ABB RAPID module: P104.mod

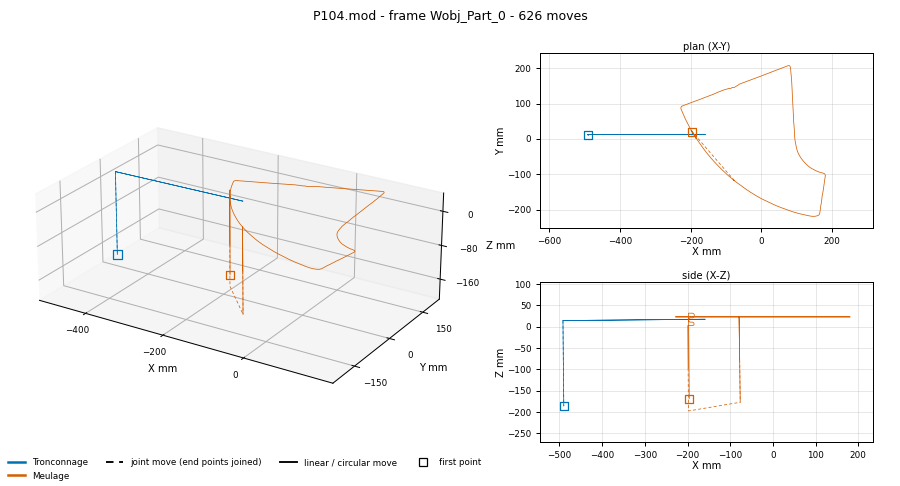
[picture p0: tool path of P104.mod in frame Wobj_Part_0, 626 of 631 moves have a stored position in this frame; points joined in program order, loops and branches not executed]
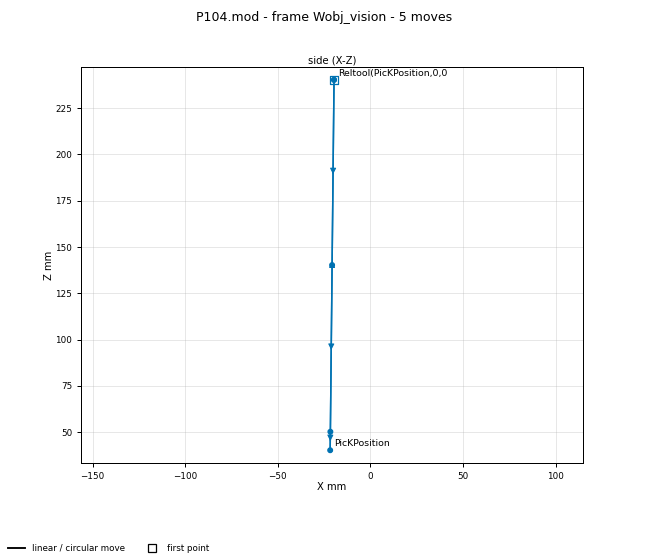
[picture p1: tool path of P104.mod in frame Wobj_vision, 5 of 631 moves have a stored position in this frame; points joined in program order, loops and branches not executed]
MODULE P104

    ! Nom         :P104
    ! Description :
    ! Créé le     :03/04/2023 16:24:55

    LOCAL CONST SPEEDDATA VitesseLente :=[10,500,0,0];
	LOCAL CONST SPEEDDATA VitesseRapide :=[30,500,0,0];
    !
    !Point de prise
    LOCAL PERS Robtarget PicKPosition := [[-21.7405517614,13.3135132251341,40.2938438381467],[-0.00337713641881813,-0.940755559571221,0.33904158472546,0.00428671346086143],[0,0,0,0],[8.999999E+09,8.999999E+09,8.999999E+09,8.999999E+09,8.999999E+09,8.999999E+09]];
	LOCAL PERS Pose Ref := [[0,0,0],[1,0,0,0]];
    !
    !Declaration des points de meulage

    !Tr_meulage_motif_1 : Meulage d'un motif
    LOCAL CONST Robtarget Tr_meulage_motif_1_0 := [[-197.52953125,22.28647265625,31.672755859375],[0.999972798976242,-0.00614910498762201,-0.0040037244179501,-0.000748335657728133],[0,0,0,0],[8.999999E+09,8.999999E+09,8.999999E+09,8.999999E+09,8.999999E+09,8.999999E+09]];
    LOCAL CONST Robtarget Tr_meulage_motif_1_1 := [[-196.9945,21.441646484375,31.672755859375],[0.999972798976242,-0.00614910498762201,-0.0040037244179501,-0.000748335657728133],[0,0,0,0],[8.999999E+09,8.999999E+09,8.999999E+09,8.999999E+09,8.999999E+09,8.999999E+09]];
    LOCAL CONST Robtarget Tr_meulage_motif_1_2 := [[-196.459453125,20.5968203125,31.6727578125],[0.999972798976242,-0.00614910498762201,-0.0040037244179501,-0.000748335657728133],[0,0,0,0],[8.999999E+09,8.999999E+09,8.999999E+09,8.999999E+09,8.999999E+09,8.999999E+09]];
    LOCAL CONST Robtarget Tr_meulage_motif_1_3 := [[-195.92440625,19.75199609375,31.6727578125],[0.999972798976242,-0.00614910498762201,-0.0040037244179501,-0.000748335657728133],[0,0,0,0],[8.999999E+09,8.999999E+09,8.999999E+09,8.999999E+09,8.999999E+09,8.999999E+09]];
    LOCAL CONST Robtarget Tr_meulage_motif_1_4 := [[-195.389375,18.907169921875,31.6727578125],[0.999972798976242,-0.00614910498762201,-0.0040037244179501,-0.000748335657728133],[0,0,0,0],[8.999999E+09,8.999999E+09,8.999999E+09,8.999999E+09,8.999999E+09,8.999999E+09]];
    LOCAL CONST Robtarget Tr_meulage_motif_1_5 := [[-194.854328125,18.06234375,31.672759765625],[0.999972798976242,-0.00614910498762201,-0.0040037244179501,-0.000748335657728133],[0,0,0,0],[8.999999E+09,8.999999E+09,8.999999E+09,8.999999E+09,8.999999E+09,8.999999E+09]];
    LOCAL CONST Robtarget Tr_meulage_motif_1_6 := [[-194.31928125,17.217517578125,31.672759765625],[0.999972798976242,-0.00614910498762201,-0.0040037244179501,-0.000748335657728133],[0,0,0,0],[8.999999E+09,8.999999E+09,8.999999E+09,8.999999E+09,8.999999E+09,8.999999E+09]];
    LOCAL CONST Robtarget Tr_meulage_motif_1_7 := [[-193.78425,16.3726923828125,31.672759765625],[0.999972798976242,-0.00614910498762201,-0.0040037244179501,-0.000748335657728133],[0,0,0,0],[8.999999E+09,8.999999E+09,8.999999E+09,8.999999E+09,8.999999E+09,8.999999E+09]];
    LOCAL CONST Robtarget Tr_meulage_motif_1_8 := [[-193.249203125,15.5278671875,31.67276171875],[0.999972798976242,-0.00614910498762201,-0.0040037244179501,-0.000748335657728133],[0,0,0,0],[8.999999E+09,8.999999E+09,8.999999E+09,8.999999E+09,8.999999E+09,8.999999E+09]];
    LOCAL CONST Robtarget Tr_meulage_motif_1_9 := [[-192.71415625,14.683041015625,31.67276171875],[0.999972798976242,-0.00614910498762201,-0.0040037244179501,-0.000748335657728133],[0,0,0,0],[8.999999E+09,8.999999E+09,8.999999E+09,8.999999E+09,8.999999E+09,8.999999E+09]];
    LOCAL CONST Robtarget Tr_meulage_motif_1_10 := [[-192.179125,13.8382158203125,31.67276171875],[0.999972798976242,-0.00614910498762201,-0.0040037244179501,-0.000748335657728133],[0,0,0,0],[8.999999E+09,8.999999E+09,8.999999E+09,8.999999E+09,8.999999E+09,8.999999E+09]];
    LOCAL CONST Robtarget Tr_meulage_motif_1_11 := [[-191.644078125,12.9933896484375,31.672763671875],[0.999972798976242,-0.00614910498762201,-0.0040037244179501,-0.000748335657728133],[0,0,0,0],[8.999999E+09,8.999999E+09,8.999999E+09,8.999999E+09,8.999999E+09,8.999999E+09]];
    LOCAL CONST Robtarget Tr_meulage_motif_1_12 := [[-191.10903125,12.148564453125,31.672763671875],[0.999972798976242,-0.00614910498762201,-0.0040037244179501,-0.000748335657728133],[0,0,0,0],[8.999999E+09,8.999999E+09,8.999999E+09,8.999999E+09,8.999999E+09,8.999999E+09]];
    LOCAL CONST Robtarget Tr_meulage_motif_1_13 := [[-190.574,11.30373828125,31.672763671875],[0.999972798976242,-0.00614910498762201,-0.0040037244179501,-0.000748335657728133],[0,0,0,0],[8.999999E+09,8.999999E+09,8.999999E+09,8.999999E+09,8.999999E+09,8.999999E+09]];
    LOCAL CONST Robtarget Tr_meulage_motif_1_14 := [[-190.038953125,10.4589130859375,31.672765625],[0.999972798976242,-0.00614910498762201,-0.0040037244179501,-0.000748335657728133],[0,0,0,0],[8.999999E+09,8.999999E+09,8.999999E+09,8.999999E+09,8.999999E+09,8.999999E+09]];
    LOCAL CONST Robtarget Tr_meulage_motif_1_15 := [[-189.50390625,9.6140869140625,31.672765625],[0.999972798976242,-0.00614910498762201,-0.0040037244179501,-0.000748335657728133],[0,0,0,0],[8.999999E+09,8.999999E+09,8.999999E+09,8.999999E+09,8.999999E+09,8.999999E+09]];
    LOCAL CONST Robtarget Tr_meulage_motif_1_16 := [[-188.968875,8.76926171875,31.672765625],[0.999972798976242,-0.00614910498762201,-0.0040037244179501,-0.000748335657728133],[0,0,0,0],[8.999999E+09,8.999999E+09,8.999999E+09,8.999999E+09,8.999999E+09,8.999999E+09]];
    LOCAL CONST Robtarget Tr_meulage_motif_1_17 := [[-188.433828125,7.92443603515625,31.672767578125],[0.999972798976242,-0.00614910498762201,-0.0040037244179501,-0.000748335657728133],[0,0,0,0],[8.999999E+09,8.999999E+09,8.999999E+09,8.999999E+09,8.999999E+09,8.999999E+09]];
    LOCAL CONST Robtarget Tr_meulage_motif_1_18 := [[-187.89878125,7.0796103515625,31.672767578125],[0.999972798976242,-0.00614910498762201,-0.0040037244179501,-0.000748335657728133],[0,0,0,0],[8.999999E+09,8.999999E+09,8.999999E+09,8.999999E+09,8.999999E+09,8.999999E+09]];
    LOCAL CONST Robtarget Tr_meulage_motif_1_19 := [[-187.368796875,6.24039208984375,31.562181640625],[0.999972798976242,-0.00614910498762201,-0.0040037244179501,-0.000748335657728133],[0,0,0,0],[8.999999E+09,8.999999E+09,8.999999E+09,8.999999E+09,8.999999E+09,8.999999E+09]];
    LOCAL CONST Robtarget Tr_meulage_motif_1_20 := [[-186.86440625,5.4394736328125,31.351009765625],[0.999972798976242,-0.00614910498762201,-0.0040037244179501,-0.000748335657728133],[0,0,0,0],[8.999999E+09,8.999999E+09,8.999999E+09,8.999999E+09,8.999999E+09,8.999999E+09]];
    LOCAL CONST Robtarget Tr_meulage_motif_1_21 := [[-186.410796875,4.71741357421875,31.07918359375],[0.999972798976242,-0.00614910498762201,-0.0040037244179501,-0.000748335657728133],[0,0,0,0],[8.999999E+09,8.999999E+09,8.999999E+09,8.999999E+09,8.999999E+09,8.999999E+09]];
    LOCAL CONST Robtarget Tr_meulage_motif_1_22 := [[-186.012203125,4.08216088867187,30.803263671875],[0.999972798976242,-0.00614910498762201,-0.0040037244179501,-0.000748335657728133],[0,0,0,0],[8.999999E+09,8.999999E+09,8.999999E+09,8.999999E+09,8.999999E+09,8.999999E+09]];
    LOCAL CONST Robtarget Tr_meulage_motif_1_23 := [[-185.42903125,3.148189453125,30.1871796875],[0.999972798976242,-0.00614910498762201,-0.0040037244179501,-0.000748335657728133],[0,0,0,0],[8.999999E+09,8.999999E+09,8.999999E+09,8.999999E+09,8.999999E+09,8.999999E+09]];
    LOCAL CONST Robtarget Tr_meulage_motif_1_24 := [[-184.88940625,2.27801293945312,29.339580078125],[0.999972798976242,-0.00614910498762201,-0.0040037244179501,-0.000748335657728133],[0,0,0,0],[8.999999E+09,8.999999E+09,8.999999E+09,8.999999E+09,8.999999E+09,8.999999E+09]];
    LOCAL CONST Robtarget Tr_meulage_motif_1_25 := [[-184.44575,1.55563366699219,28.315771484375],[0.999972798976242,-0.00614910498762201,-0.0040037244179501,-0.000748335657728133],[0,0,0,0],[8.999999E+09,8.999999E+09,8.999999E+09,8.999999E+09,8.999999E+09,8.999999E+09]];
    LOCAL CONST Robtarget Tr_meulage_motif_1_26 := [[-184.195328125,1.13640502929688,27.199658203125],[0.999972798976242,-0.00614910498762201,-0.0040037244179501,-0.000748335657728133],[0,0,0,0],[8.999999E+09,8.999999E+09,8.999999E+09,8.999999E+09,8.999999E+09,8.999999E+09]];
    LOCAL CONST Robtarget Tr_meulage_motif_1_27 := [[-184.187578125,1.10928845214844,26.503734375],[0.999972798976242,-0.00614910498762201,-0.0040037244179501,-0.000748335657728133],[0,0,0,0],[8.999999E+09,8.999999E+09,8.999999E+09,8.999999E+09,8.999999E+09,8.999999E+09]];
    LOCAL CONST Robtarget Tr_meulage_motif_1_28 := [[-184.193953125,1.10524719238281,25.84252734375],[0.999972798976242,-0.00614910498762201,-0.0040037244179501,-0.000748335657728133],[0,0,0,0],[8.999999E+09,8.999999E+09,8.999999E+09,8.999999E+09,8.999999E+09,8.999999E+09]];
    LOCAL CONST Robtarget Tr_meulage_motif_1_29 := [[-184.2296875,1.14756665039062,25.1814765625],[0.999972798976242,-0.00614910498762201,-0.0040037244179501,-0.000748335657728133],[0,0,0,0],[8.999999E+09,8.999999E+09,8.999999E+09,8.999999E+09,8.999999E+09,8.999999E+09]];
    LOCAL CONST Robtarget Tr_meulage_motif_1_30 := [[-184.506890625,1.5617412109375,24.079798828125],[0.999972798976242,-0.00614910498762201,-0.0040037244179501,-0.000748335657728133],[0,0,0,0],[8.999999E+09,8.999999E+09,8.999999E+09,8.999999E+09,8.999999E+09,8.999999E+09]];
    LOCAL CONST Robtarget Tr_meulage_motif_1_31 := [[-184.9749375,2.27928784179687,23.07323828125],[0.999972798976242,-0.00614910498762201,-0.0040037244179501,-0.000748335657728133],[0,0,0,0],[8.999999E+09,8.999999E+09,8.999999E+09,8.999999E+09,8.999999E+09,8.999999E+09]];
    LOCAL CONST Robtarget Tr_meulage_motif_1_32 := [[-185.5305,3.13882202148437,22.24441796875],[0.999972798976242,-0.00614910498762201,-0.0040037244179501,-0.000748335657728133],[0,0,0,0],[8.999999E+09,8.999999E+09,8.999999E+09,8.999999E+09,8.999999E+09,8.999999E+09]];
    LOCAL CONST Robtarget Tr_meulage_motif_1_33 := [[-185.9019375,3.71687768554688,21.848693359375],[0.999972798976242,-0.00614910498762201,-0.0040037244179501,-0.000748335657728133],[0,0,0,0],[8.999999E+09,8.999999E+09,8.999999E+09,8.999999E+09,8.999999E+09,8.999999E+09]];
    LOCAL CONST Robtarget Tr_meulage_motif_1_34 := [[-186.526296875,4.69233837890625,21.36119140625],[0.999972798976242,-0.00614910498762201,-0.0040037244179501,-0.000748335657728133],[0,0,0,0],[8.999999E+09,8.999999E+09,8.999999E+09,8.999999E+09,8.999999E+09,8.999999E+09]];
    LOCAL CONST Robtarget Tr_meulage_motif_1_35 := [[-186.980984375,5.40462841796875,21.097115234375],[0.999972798976242,-0.00614910498762201,-0.0040037244179501,-0.000748335657728133],[0,0,0,0],[8.999999E+09,8.999999E+09,8.999999E+09,8.999999E+09,8.999999E+09,8.999999E+09]];
    LOCAL CONST Robtarget Tr_meulage_motif_1_36 := [[-187.481609375,6.19075634765625,20.89266015625],[0.999972798976242,-0.00614910498762201,-0.0040037244179501,-0.000748335657728133],[0,0,0,0],[8.999999E+09,8.999999E+09,8.999999E+09,8.999999E+09,8.999999E+09,8.999999E+09]];
    LOCAL CONST Robtarget Tr_meulage_motif_1_37 := [[-188.007828125,7.019341796875,20.784072265625],[0.999972798976242,-0.00614910498762201,-0.0040037244179501,-0.000748335657728133],[0,0,0,0],[8.999999E+09,8.999999E+09,8.999999E+09,8.999999E+09,8.999999E+09,8.999999E+09]];
    LOCAL CONST Robtarget Tr_meulage_motif_1_38 := [[-188.53996875,7.8572080078125,20.673484375],[0.999972798976242,-0.00614910498762201,-0.0040037244179501,-0.000748335657728133],[0,0,0,0],[8.999999E+09,8.999999E+09,8.999999E+09,8.999999E+09,8.999999E+09,8.999999E+09]];
    LOCAL CONST Robtarget Tr_meulage_motif_1_39 := [[-189.075,8.7020341796875,20.673484375],[0.999972798976242,-0.00614910498762201,-0.0040037244179501,-0.000748335657728133],[0,0,0,0],[8.999999E+09,8.999999E+09,8.999999E+09,8.999999E+09,8.999999E+09,8.999999E+09]];
    LOCAL CONST Robtarget Tr_meulage_motif_1_40 := [[-189.610046875,9.546859375,20.673482421875],[0.999972798976242,-0.00614910498762201,-0.0040037244179501,-0.000748335657728133],[0,0,0,0],[8.999999E+09,8.999999E+09,8.999999E+09,8.999999E+09,8.999999E+09,8.999999E+09]];
    LOCAL CONST Robtarget Tr_meulage_motif_1_41 := [[-190.14509375,10.391685546875,20.673482421875],[0.999972798976242,-0.00614910498762201,-0.0040037244179501,-0.000748335657728133],[0,0,0,0],[8.999999E+09,8.999999E+09,8.999999E+09,8.999999E+09,8.999999E+09,8.999999E+09]];
    LOCAL CONST Robtarget Tr_meulage_motif_1_42 := [[-190.680125,11.2365107421875,20.673482421875],[0.999972798976242,-0.00614910498762201,-0.0040037244179501,-0.000748335657728133],[0,0,0,0],[8.999999E+09,8.999999E+09,8.999999E+09,8.999999E+09,8.999999E+09,8.999999E+09]];
    LOCAL CONST Robtarget Tr_meulage_motif_1_43 := [[-191.215171875,12.0813369140625,20.67348046875],[0.999972798976242,-0.00614910498762201,-0.0040037244179501,-0.000748335657728133],[0,0,0,0],[8.999999E+09,8.999999E+09,8.999999E+09,8.999999E+09,8.999999E+09,8.999999E+09]];
    LOCAL CONST Robtarget Tr_meulage_motif_1_44 := [[-191.75021875,12.926162109375,20.67348046875],[0.999972798976242,-0.00614910498762201,-0.0040037244179501,-0.000748335657728133],[0,0,0,0],[8.999999E+09,8.999999E+09,8.999999E+09,8.999999E+09,8.999999E+09,8.999999E+09]];
    LOCAL CONST Robtarget Tr_meulage_motif_1_45 := [[-192.28525,13.77098828125,20.67348046875],[0.999972798976242,-0.00614910498762201,-0.0040037244179501,-0.000748335657728133],[0,0,0,0],[8.999999E+09,8.999999E+09,8.999999E+09,8.999999E+09,8.999999E+09,8.999999E+09]];
    LOCAL CONST Robtarget Tr_meulage_motif_1_46 := [[-192.820296875,14.6158134765625,20.673478515625],[0.999972798976242,-0.00614910498762201,-0.0040037244179501,-0.000748335657728133],[0,0,0,0],[8.999999E+09,8.999999E+09,8.999999E+09,8.999999E+09,8.999999E+09,8.999999E+09]];
    LOCAL CONST Robtarget Tr_meulage_motif_1_47 := [[-193.35534375,15.4606396484375,20.673478515625],[0.999972798976242,-0.00614910498762201,-0.0040037244179501,-0.000748335657728133],[0,0,0,0],[8.999999E+09,8.999999E+09,8.999999E+09,8.999999E+09,8.999999E+09,8.999999E+09]];
    LOCAL CONST Robtarget Tr_meulage_motif_1_48 := [[-193.890375,16.30546484375,20.673478515625],[0.999972798976242,-0.00614910498762201,-0.0040037244179501,-0.000748335657728133],[0,0,0,0],[8.999999E+09,8.999999E+09,8.999999E+09,8.999999E+09,8.999999E+09,8.999999E+09]];
    LOCAL CONST Robtarget Tr_meulage_motif_1_49 := [[-194.422515625,17.14333203125,20.562890625],[0.999972798976242,-0.00614910498762201,-0.0040037244179501,-0.000748335657728133],[0,0,0,0],[8.999999E+09,8.999999E+09,8.999999E+09,8.999999E+09,8.999999E+09,8.999999E+09]];
    LOCAL CONST Robtarget Tr_meulage_motif_1_50 := [[-194.93096875,17.94166796875,20.351716796875],[0.999972798976242,-0.00614910498762201,-0.0040037244179501,-0.000748335657728133],[0,0,0,0],[8.999999E+09,8.999999E+09,8.999999E+09,8.999999E+09,8.999999E+09,8.999999E+09]];
    LOCAL CONST Robtarget Tr_meulage_motif_1_51 := [[-195.389828125,18.66040625,20.079890625],[0.999972798976242,-0.00614910498762201,-0.0040037244179501,-0.000748335657728133],[0,0,0,0],[8.999999E+09,8.999999E+09,8.999999E+09,8.999999E+09,8.999999E+09,8.999999E+09]];
    LOCAL CONST Robtarget Tr_meulage_motif_1_52 := [[-195.7734375,19.259640625,19.77575390625],[0.999972798976242,-0.00614910498762201,-0.0040037244179501,-0.000748335657728133],[0,0,0,0],[8.999999E+09,8.999999E+09,8.999999E+09,8.999999E+09,8.999999E+09,8.999999E+09]];
    LOCAL CONST Robtarget Tr_meulage_motif_1_53 := [[-196.333328125,20.129537109375,19.113263671875],[0.999972798976242,-0.00614910498762201,-0.0040037244179501,-0.000748335657728133],[0,0,0,0],[8.999999E+09,8.999999E+09,8.999999E+09,8.999999E+09,8.999999E+09,8.999999E+09]];
    LOCAL CONST Robtarget Tr_meulage_motif_1_54 := [[-196.82459375,20.88600390625,18.211384765625],[0.999972798976242,-0.00614910498762201,-0.0040037244179501,-0.000748335657728133],[0,0,0,0],[8.999999E+09,8.999999E+09,8.999999E+09,8.999999E+09,8.999999E+09,8.999999E+09]];
    LOCAL CONST Robtarget Tr_meulage_motif_1_55 := [[-197.120921875,21.33156640625,17.165421875],[0.999972798976242,-0.00614910498762201,-0.0040037244179501,-0.000748335657728133],[0,0,0,0],[8.999999E+09,8.999999E+09,8.999999E+09,8.999999E+09,8.999999E+09,8.999999E+09]];
    LOCAL CONST Robtarget Tr_meulage_motif_1_56 := [[-197.22646875,21.4834375,16.472248046875],[0.999972798976242,-0.00614910498762201,-0.0040037244179501,-0.000748335657728133],[0,0,0,0],[8.999999E+09,8.999999E+09,8.999999E+09,8.999999E+09,8.999999E+09,8.999999E+09]];
    LOCAL CONST Robtarget Tr_meulage_motif_1_57 := [[-197.2680625,21.532669921875,15.7022978515625],[0.999972798976242,-0.00614910498762201,-0.0040037244179501,-0.000748335657728133],[0,0,0,0],[8.999999E+09,8.999999E+09,8.999999E+09,8.999999E+09,8.999999E+09,8.999999E+09]];
    LOCAL CONST Robtarget Tr_meulage_motif_1_58 := [[-197.239671875,21.4714140625,14.9324736328125],[0.999972798976242,-0.00614910498762201,-0.0040037244179501,-0.000748335657728133],[0,0,0,0],[8.999999E+09,8.999999E+09,8.999999E+09,8.999999E+09,8.999999E+09,8.999999E+09]];
    LOCAL CONST Robtarget Tr_meulage_motif_1_59 := [[-197.025875,21.11015625,13.8242958984375],[0.999972798976242,-0.00614910498762201,-0.0040037244179501,-0.000748335657728133],[0,0,0,0],[8.999999E+09,8.999999E+09,8.999999E+09,8.999999E+09,8.999999E+09,8.999999E+09]];
    LOCAL CONST Robtarget Tr_meulage_motif_1_60 := [[-196.80984375,20.7565546875,13.238646484375],[0.999972798976242,-0.00614910498762201,-0.0040037244179501,-0.000748335657728133],[0,0,0,0],[8.999999E+09,8.999999E+09,8.999999E+09,8.999999E+09,8.999999E+09,8.999999E+09]];
    LOCAL CONST Robtarget Tr_meulage_motif_1_61 := [[-196.343765625,20.00166796875,12.351580078125],[0.999972798976242,-0.00614910498762201,-0.0040037244179501,-0.000748335657728133],[0,0,0,0],[8.999999E+09,8.999999E+09,8.999999E+09,8.999999E+09,8.999999E+09,8.999999E+09]];
    LOCAL CONST Robtarget Tr_meulage_motif_1_62 := [[-196.034390625,19.50433203125,11.937294921875],[0.999972798976242,-0.00614910498762201,-0.0040037244179501,-0.000748335657728133],[0,0,0,0],[8.999999E+09,8.999999E+09,8.999999E+09,8.999999E+09,8.999999E+09,8.999999E+09]];
    LOCAL CONST Robtarget Tr_meulage_motif_1_63 := [[-195.441515625,18.5565703125,11.39323828125],[0.999972798976242,-0.00614910498762201,-0.0040037244179501,-0.000748335657728133],[0,0,0,0],[8.999999E+09,8.999999E+09,8.999999E+09,8.999999E+09,8.999999E+09,8.999999E+09]];
    LOCAL CONST Robtarget Tr_meulage_motif_1_64 := [[-195.002640625,17.85728125,11.0977578125],[0.999972798976242,-0.00614910498762201,-0.0040037244179501,-0.000748335657728133],[0,0,0,0],[8.999999E+09,8.999999E+09,8.999999E+09,8.999999E+09,8.999999E+09,8.999999E+09]];
    LOCAL CONST Robtarget Tr_meulage_motif_1_65 := [[-194.505953125,17.068654296875,10.893302734375],[0.999972798976242,-0.00614910498762201,-0.0040037244179501,-0.000748335657728133],[0,0,0,0],[8.999999E+09,8.999999E+09,8.999999E+09,8.999999E+09,8.999999E+09,8.999999E+09]];
    LOCAL CONST Robtarget Tr_meulage_motif_1_66 := [[-193.981828125,16.2387412109375,10.784716796875],[0.999972798976242,-0.00614910498762201,-0.0040037244179501,-0.000748335657728133],[0,0,0,0],[8.999999E+09,8.999999E+09,8.999999E+09,8.999999E+09,8.999999E+09,8.999999E+09]];
    LOCAL CONST Robtarget Tr_meulage_motif_1_67 := [[-193.451828125,15.3995234375,10.674130859375],[0.999972798976242,-0.00614910498762201,-0.0040037244179501,-0.000748335657728133],[0,0,0,0],[8.999999E+09,8.999999E+09,8.999999E+09,8.999999E+09,8.999999E+09,8.999999E+09]];
    LOCAL CONST Robtarget Tr_meulage_motif_1_68 := [[-192.91678125,14.554697265625,10.6741318359375],[0.999972798976242,-0.00614910498762201,-0.0040037244179501,-0.000748335657728133],[0,0,0,0],[8.999999E+09,8.999999E+09,8.999999E+09,8.999999E+09,8.999999E+09,8.999999E+09]];
    LOCAL CONST Robtarget Tr_meulage_motif_1_69 := [[-192.38175,13.7098720703125,10.6741318359375],[0.999972798976242,-0.00614910498762201,-0.0040037244179501,-0.000748335657728133],[0,0,0,0],[8.999999E+09,8.999999E+09,8.999999E+09,8.999999E+09,8.999999E+09,8.999999E+09]];
    LOCAL CONST Robtarget Tr_meulage_motif_1_70 := [[-191.846703125,12.8650458984375,10.6741328125],[0.999972798976242,-0.00614910498762201,-0.0040037244179501,-0.000748335657728133],[0,0,0,0],[8.999999E+09,8.999999E+09,8.999999E+09,8.999999E+09,8.999999E+09,8.999999E+09]];
    LOCAL CONST Robtarget Tr_meulage_motif_1_71 := [[-191.31165625,12.020220703125,10.6741337890625],[0.999972798976242,-0.00614910498762201,-0.0040037244179501,-0.000748335657728133],[0,0,0,0],[8.999999E+09,8.999999E+09,8.999999E+09,8.999999E+09,8.999999E+09,8.999999E+09]];
    LOCAL CONST Robtarget Tr_meulage_motif_1_72 := [[-190.776625,11.17539453125,10.674134765625],[0.999972798976242,-0.00614910498762201,-0.0040037244179501,-0.000748335657728133],[0,0,0,0],[8.999999E+09,8.999999E+09,8.999999E+09,8.999999E+09,8.999999E+09,8.999999E+09]];
    LOCAL CONST Robtarget Tr_meulage_motif_1_73 := [[-190.241578125,10.3305693359375,10.674134765625],[0.999972798976242,-0.00614910498762201,-0.0040037244179501,-0.000748335657728133],[0,0,0,0],[8.999999E+09,8.999999E+09,8.999999E+09,8.999999E+09,8.999999E+09,8.999999E+09]];
    LOCAL CONST Robtarget Tr_meulage_motif_1_74 := [[-189.70653125,9.4857431640625,10.6741357421875],[0.999972798976242,-0.00614910498762201,-0.0040037244179501,-0.000748335657728133],[0,0,0,0],[8.999999E+09,8.999999E+09,8.999999E+09,8.999999E+09,8.999999E+09,8.999999E+09]];
    LOCAL CONST Robtarget Tr_meulage_motif_1_75 := [[-189.1715,8.64091796875,10.67413671875],[0.999972798976242,-0.00614910498762201,-0.0040037244179501,-0.000748335657728133],[0,0,0,0],[8.999999E+09,8.999999E+09,8.999999E+09,8.999999E+09,8.999999E+09,8.999999E+09]];
    LOCAL CONST Robtarget Tr_meulage_motif_1_76 := [[-188.636453125,7.79609228515625,10.67413671875],[0.999972798976242,-0.00614910498762201,-0.0040037244179501,-0.000748335657728133],[0,0,0,0],[8.999999E+09,8.999999E+09,8.999999E+09,8.999999E+09,8.999999E+09,8.999999E+09]];
    LOCAL CONST Robtarget Tr_meulage_motif_1_77 := [[-188.10140625,6.9512666015625,10.6741376953125],[0.999972798976242,-0.00614910498762201,-0.0040037244179501,-0.000748335657728133],[0,0,0,0],[8.999999E+09,8.999999E+09,8.999999E+09,8.999999E+09,8.999999E+09,8.999999E+09]];
    LOCAL CONST Robtarget Tr_meulage_motif_1_78 := [[-187.571421875,6.11204833984375,10.5635517578125],[0.999972798976242,-0.00614910498762201,-0.0040037244179501,-0.000748335657728133],[0,0,0,0],[8.999999E+09,8.999999E+09,8.999999E+09,8.999999E+09,8.999999E+09,8.999999E+09]];
    LOCAL CONST Robtarget Tr_meulage_motif_1_79 := [[-187.06703125,5.31113037109375,10.35237890625],[0.999972798976242,-0.00614910498762201,-0.0040037244179501,-0.000748335657728133],[0,0,0,0],[8.999999E+09,8.999999E+09,8.999999E+09,8.999999E+09,8.999999E+09,8.999999E+09]];
    LOCAL CONST Robtarget Tr_meulage_motif_1_80 := [[-186.613421875,4.58906982421875,10.080552734375],[0.999972798976242,-0.00614910498762201,-0.0040037244179501,-0.000748335657728133],[0,0,0,0],[8.999999E+09,8.999999E+09,8.999999E+09,8.999999E+09,8.999999E+09,8.999999E+09]];
    LOCAL CONST Robtarget Tr_meulage_motif_1_81 := [[-186.214828125,3.95381713867188,9.8046337890625],[0.999972798976242,-0.00614910498762201,-0.0040037244179501,-0.000748335657728133],[0,0,0,0],[8.999999E+09,8.999999E+09,8.999999E+09,8.999999E+09,8.999999E+09,8.999999E+09]];
    LOCAL CONST Robtarget Tr_meulage_motif_1_82 := [[-185.631671875,3.019845703125,9.1885498046875],[0.999972798976242,-0.00614910498762201,-0.0040037244179501,-0.000748335657728133],[0,0,0,0],[8.999999E+09,8.999999E+09,8.999999E+09,8.999999E+09,8.999999E+09,8.999999E+09]];
    LOCAL CONST Robtarget Tr_meulage_motif_1_83 := [[-185.12840625,2.20612158203125,8.294640625],[0.999972798976242,-0.00614910498762201,-0.0040037244179501,-0.000748335657728133],[0,0,0,0],[8.999999E+09,8.999999E+09,8.999999E+09,8.999999E+09,8.999999E+09,8.999999E+09]];
    LOCAL CONST Robtarget Tr_meulage_motif_1_84 := [[-184.812984375,1.68488000488281,7.20871142578125],[0.999972798976242,-0.00614910498762201,-0.0040037244179501,-0.000748335657728133],[0,0,0,0],[8.999999E+09,8.999999E+09,8.999999E+09,8.999999E+09,8.999999E+09,8.999999E+09]];
    LOCAL CONST Robtarget Tr_meulage_motif_1_85 := [[-184.731890625,1.53582434082031,6.22440087890625],[0.999972798976242,-0.00614910498762201,-0.0040037244179501,-0.000748335657728133],[0,0,0,0],[8.999999E+09,8.999999E+09,8.999999E+09,8.999999E+09,8.999999E+09,8.999999E+09]];
    LOCAL CONST Robtarget Tr_meulage_motif_1_86 := [[-184.804203125,1.64564172363281,6.0197578125],[0.999972798976242,-0.00614910498762201,-0.0040037244179501,-0.000748335657728133],[0,0,0,0],[8.999999E+09,8.999999E+09,8.999999E+09,8.999999E+09,8.999999E+09,8.999999E+09]];
    LOCAL CONST Robtarget Tr_meulage_motif_1_87 := [[-184.87721875,1.7454326171875,5.29339892578125],[0.999972798976242,-0.00614910498762201,-0.0040037244179501,-0.000748335657728133],[0,0,0,0],[8.999999E+09,8.999999E+09,8.999999E+09,8.999999E+09,8.999999E+09,8.999999E+09]];
    LOCAL CONST Robtarget Tr_meulage_motif_1_88 := [[-185.252234375,2.3175673828125,4.35655322265625],[0.999972798976242,-0.00614910498762201,-0.0040037244179501,-0.000748335657728133],[0,0,0,0],[8.999999E+09,8.999999E+09,8.999999E+09,8.999999E+09,8.999999E+09,8.999999E+09]];
    LOCAL CONST Robtarget Tr_meulage_motif_1_89 := [[-185.5550625,2.78582861328125,3.89277075195313],[0.999972798976242,-0.00614910498762201,-0.0040037244179501,-0.000748335657728133],[0,0,0,0],[8.999999E+09,8.999999E+09,8.999999E+09,8.999999E+09,8.999999E+09,8.999999E+09]];
    LOCAL CONST Robtarget Tr_meulage_motif_1_90 := [[-186.1649375,3.73750390625,3.3623671875],[0.999972798976242,-0.00614910498762201,-0.0040037244179501,-0.000748335657728133],[0,0,0,0],[8.999999E+09,8.999999E+09,8.999999E+09,8.999999E+09,8.999999E+09,8.999999E+09]];
    LOCAL CONST Robtarget Tr_meulage_motif_1_91 := [[-186.619625,4.4497939453125,3.0982900390625],[0.999972798976242,-0.00614910498762201,-0.0040037244179501,-0.000748335657728133],[0,0,0,0],[8.999999E+09,8.999999E+09,8.999999E+09,8.999999E+09,8.999999E+09,8.999999E+09]];
    LOCAL CONST Robtarget Tr_meulage_motif_1_92 := [[-187.12025,5.235921875,2.893833984375],[0.999972798976242,-0.00614910498762201,-0.0040037244179501,-0.000748335657728133],[0,0,0,0],[8.999999E+09,8.999999E+09,8.999999E+09,8.999999E+09,8.999999E+09,8.999999E+09]];
    LOCAL CONST Robtarget Tr_meulage_motif_1_93 := [[-187.64646875,6.06450732421875,2.78524658203125],[0.999972798976242,-0.00614910498762201,-0.0040037244179501,-0.000748335657728133],[0,0,0,0],[8.999999E+09,8.999999E+09,8.999999E+09,8.999999E+09,8.999999E+09,8.999999E+09]];
    LOCAL CONST Robtarget Tr_meulage_motif_1_94 := [[-188.178609375,6.90237353515625,2.67465942382813],[0.999972798976242,-0.00614910498762201,-0.0040037244179501,-0.000748335657728133],[0,0,0,0],[8.999999E+09,8.999999E+09,8.999999E+09,8.999999E+09,8.999999E+09,8.999999E+09]];
    LOCAL CONST Robtarget Tr_meulage_motif_1_95 := [[-188.713640625,7.74719921875,2.67465869140625],[0.999972798976242,-0.00614910498762201,-0.0040037244179501,-0.000748335657728133],[0,0,0,0],[8.999999E+09,8.999999E+09,8.999999E+09,8.999999E+09,8.999999E+09,8.999999E+09]];
    LOCAL CONST Robtarget Tr_meulage_motif_1_96 := [[-189.2486875,8.592025390625,2.674658203125],[0.999972798976242,-0.00614910498762201,-0.0040037244179501,-0.000748335657728133],[0,0,0,0],[8.999999E+09,8.999999E+09,8.999999E+09,8.999999E+09,8.999999E+09,8.999999E+09]];
    LOCAL CONST Robtarget Tr_meulage_motif_1_97 := [[-189.783734375,9.4368505859375,2.67465747070313],[0.999972798976242,-0.00614910498762201,-0.0040037244179501,-0.000748335657728133],[0,0,0,0],[8.999999E+09,8.999999E+09,8.999999E+09,8.999999E+09,8.999999E+09,8.999999E+09]];
    LOCAL CONST Robtarget Tr_meulage_motif_1_98 := [[-190.318765625,10.2816767578125,2.67465673828125],[0.999972798976242,-0.00614910498762201,-0.0040037244179501,-0.000748335657728133],[0,0,0,0],[8.999999E+09,8.999999E+09,8.999999E+09,8.999999E+09,8.999999E+09,8.999999E+09]];
    LOCAL CONST Robtarget Tr_meulage_motif_1_99 := [[-190.8538125,11.126501953125,2.67465600585937],[0.999972798976242,-0.00614910498762201,-0.0040037244179501,-0.000748335657728133],[0,0,0,0],[8.999999E+09,8.999999E+09,8.999999E+09,8.999999E+09,8.999999E+09,8.999999E+09]];
    LOCAL CONST Robtarget Tr_meulage_motif_1_100 := [[-191.388859375,11.971328125,2.67465551757813],[0.999972798976242,-0.00614910498762201,-0.0040037244179501,-0.000748335657728133],[0,0,0,0],[8.999999E+09,8.999999E+09,8.999999E+09,8.999999E+09,8.999999E+09,8.999999E+09]];
    LOCAL CONST Robtarget Tr_meulage_motif_1_101 := [[-191.923890625,12.8161533203125,2.67465478515625],[0.999972798976242,-0.00614910498762201,-0.0040037244179501,-0.000748335657728133],[0,0,0,0],[8.999999E+09,8.999999E+09,8.999999E+09,8.999999E+09,8.999999E+09,8.999999E+09]];
    LOCAL CONST Robtarget Tr_meulage_motif_1_102 := [[-192.4589375,13.6609794921875,2.67465405273437],[0.999972798976242,-0.00614910498762201,-0.0040037244179501,-0.000748335657728133],[0,0,0,0],[8.999999E+09,8.999999E+09,8.999999E+09,8.999999E+09,8.999999E+09,8.999999E+09]];
    LOCAL CONST Robtarget Tr_meulage_motif_1_103 := [[-192.993984375,14.5058046875,2.67465356445312],[0.999972798976242,-0.00614910498762201,-0.0040037244179501,-0.000748335657728133],[0,0,0,0],[8.999999E+09,8.999999E+09,8.999999E+09,8.999999E+09,8.999999E+09,8.999999E+09]];
    LOCAL CONST Robtarget Tr_meulage_motif_1_104 := [[-193.529015625,15.350630859375,2.67465283203125],[0.999972798976242,-0.00614910498762201,-0.0040037244179501,-0.000748335657728133],[0,0,0,0],[8.999999E+09,8.999999E+09,8.999999E+09,8.999999E+09,8.999999E+09,8.999999E+09]];
    LOCAL CONST Robtarget Tr_meulage_motif_1_105 := [[-194.0640625,16.1954560546875,2.67465209960938],[0.999972798976242,-0.00614910498762201,-0.0040037244179501,-0.000748335657728133],[0,0,0,0],[8.999999E+09,8.999999E+09,8.999999E+09,8.999999E+09,8.999999E+09,8.999999E+09]];
    LOCAL CONST Robtarget Tr_meulage_motif_1_106 := [[-194.599109375,17.04028125,2.6746513671875],[0.999972798976242,-0.00614910498762201,-0.0040037244179501,-0.000748335657728133],[0,0,0,0],[8.999999E+09,8.999999E+09,8.999999E+09,8.999999E+09,8.999999E+09,8.999999E+09]];
    LOCAL CONST Robtarget Tr_meulage_motif_1_107 := [[-195.134140625,17.885107421875,2.67465087890625],[0.999972798976242,-0.00614910498762201,-0.0040037244179501,-0.000748335657728133],[0,0,0,0],[8.999999E+09,8.999999E+09,8.999999E+09,8.999999E+09,8.999999E+09,8.999999E+09]];
    LOCAL CONST Robtarget Tr_meulage_motif_1_108 := [[-195.6691875,18.72993359375,2.67465014648438],[0.999972798976242,-0.00614910498762201,-0.0040037244179501,-0.000748335657728133],[0,0,0,0],[8.999999E+09,8.999999E+09,8.999999E+09,8.999999E+09,8.999999E+09,8.999999E+09]];
    LOCAL CONST Robtarget Tr_meulage_motif_1_109 := [[-196.204234375,19.574759765625,2.6746494140625],[0.999972798976242,-0.00614910498762201,-0.0040037244179501,-0.000748335657728133],[0,0,0,0],[8.999999E+09,8.999999E+09,8.999999E+09,8.999999E+09,8.999999E+09,8.999999E+09]];
    LOCAL CONST Robtarget Tr_meulage_motif_1_110 := [[-196.739265625,20.419583984375,2.67464868164063],[0.999972798976242,-0.00614910498762201,-0.0040037244179501,-0.000748335657728133],[0,0,0,0],[8.999999E+09,8.999999E+09,8.999999E+09,8.999999E+09,8.999999E+09,8.999999E+09]];
    LOCAL CONST Robtarget Tr_meulage_motif_1_111 := [[-197.2743125,21.26441015625,2.67464819335938],[0.999972798976242,-0.00614910498762201,-0.0040037244179501,-0.000748335657728133],[0,0,0,0],[8.999999E+09,8.999999E+09,8.999999E+09,8.999999E+09,8.999999E+09,8.999999E+09]];
    LOCAL CONST Robtarget Tr_meulage_motif_1_112 := [[-197.809359375,22.109236328125,2.6746474609375],[0.999972798976242,-0.00614910498762201,-0.0040037244179501,-0.000748335657728133],[0,0,0,0],[8.999999E+09,8.999999E+09,8.999999E+09,8.999999E+09,8.999999E+09,8.999999E+09]];
    LOCAL CONST Robtarget Tr_meulage_motif_1_113 := [[-198.344390625,22.9540625,2.67464672851563],[0.999972798976242,-0.00614910498762201,-0.0040037244179501,-0.000748335657728133],[0,0,0,0],[8.999999E+09,8.999999E+09,8.999999E+09,8.999999E+09,8.999999E+09,8.999999E+09]];
    LOCAL CONST Robtarget Tr_meulage_motif_1_114 := [[-198.8794375,23.79888671875,2.67464624023438],[0.999972798976242,-0.00614910498762201,-0.0040037244179501,-0.000748335657728133],[0,0,0,0],[8.999999E+09,8.999999E+09,8.999999E+09,8.999999E+09,8.999999E+09,8.999999E+09]];
    LOCAL CONST Robtarget Tr_meulage_motif_1_115 := [[-199.414484375,24.643712890625,2.6746455078125],[0.999972798976242,-0.00614910498762201,-0.0040037244179501,-0.000748335657728133],[0,0,0,0],[8.999999E+09,8.999999E+09,8.999999E+09,8.999999E+09,8.999999E+09,8.999999E+09]];

    !Tr_meulage_bavure : Meulage de la bavure
    LOCAL CONST Robtarget Tr_meulage_bavure_0 := [[-79.2966015625,-115.933734375,23],[0.999962044987152,-0.00548384724755965,-0.00674103072583157,0.000628099698816427],[0,0,0,0],[8.999999E+09,8.999999E+09,8.999999E+09,8.999999E+09,8.999999E+09,8.999999E+09]];
    LOCAL CONST Robtarget Tr_meulage_bavure_1 := [[-85.8425,-110.82015625,23],[0.999962056853819,-0.00549252218275107,-0.00673231579668442,0.000626878589757369],[0,0,0,0],[8.999999E+09,8.999999E+09,8.999999E+09,8.999999E+09,8.999999E+09,8.999999E+09]];
    LOCAL CONST Robtarget Tr_meulage_bavure_2 := [[-86.521640625,-110.2841484375,23],[0.999962091769832,-0.0055166983173104,-0.00670768574567177,0.000622908432619115],[0,0,0,0],[8.999999E+09,8.999999E+09,8.999999E+09,8.999999E+09,8.999999E+09,8.999999E+09]];
    LOCAL CONST Robtarget Tr_meulage_bavure_3 := [[-86.9234296875,-109.95715625,23],[0.999962145327792,-0.00555203521865422,-0.00667105130281792,0.000616352890767744],[0,0,0,0],[8.999999E+09,8.999999E+09,8.999999E+09,8.999999E+09,8.999999E+09,8.999999E+09]];
    LOCAL CONST Robtarget Tr_meulage_bavure_4 := [[-90.2432265625,-107.1154921875,23],[0.999962210186898,-0.00559318697490386,-0.00662762652041128,0.000607473706764753],[0,0,0,0],[8.999999E+09,8.999999E+09,8.999999E+09,8.999999E+09,8.999999E+09,8.999999E+09]];
    LOCAL CONST Robtarget Tr_meulage_bavure_5 := [[-91.8843359375,-105.69653125,23],[0.999962276745104,-0.00563602581142986,-0.00658213997689869,0.000596433671751232],[0,0,0,0],[8.999999E+09,8.999999E+09,8.999999E+09,8.999999E+09,8.999999E+09,8.999999E+09]];
    LOCAL CONST Robtarget Tr_meulage_bavure_6 := [[-91.9569375,-105.614515625,23],[0.999962333392572,-0.00567909898670531,-0.00653751786602696,0.00058351600901736],[0,0,0,0],[8.999999E+09,8.999999E+09,8.999999E+09,8.999999E+09,8.999999E+09,8.999999E+09]];
    LOCAL CONST Robtarget Tr_meulage_bavure_7 := [[-93.0571015625,-104.660140625,23],[0.999962369534406,-0.00572333347124117,-0.00649455366529783,0.000568983130320225],[0,0,0,0],[8.999999E+09,8.999999E+09,8.999999E+09,8.999999E+09,8.999999E+09,8.999999E+09]];
    LOCAL CONST Robtarget Tr_meulage_bavure_8 := [[-99.2814921875,-98.96675,23],[0.999962377126769,-0.00577096308388516,-0.00645246842950749,0.00055314304883965],[0,0,0,0],[8.999999E+09,8.999999E+09,8.999999E+09,8.999999E+09,8.999999E+09,8.999999E+09]];
    LOCAL CONST Robtarget Tr_meulage_bavure_9 := [[-102.1833828125,-96.3584609375,23],[0.999962352956623,-0.00582351918060984,-0.00641027247403132,0.000536377308094372],[0,0,0,0],[8.999999E+09,8.999999E+09,8.999999E+09,8.999999E+09,8.999999E+09,8.999999E+09]];
    LOCAL CONST Robtarget Tr_meulage_bavure_10 := [[-103.9701875,-94.720625,23],[0.99996229984397,-0.00588047724891152,-0.00636785334858952,0.000518962247058902],[0,0,0,0],[8.999999E+09,8.999999E+09,8.999999E+09,8.999999E+09,8.999999E+09,8.999999E+09]];
    LOCAL CONST Robtarget Tr_meulage_bavure_11 := [[-107.26690625,-91.5796484375,23],[0.999962225811715,-0.00593927655434447,-0.00632617877522439,0.000501403825998657],[0,0,0,0],[8.999999E+09,8.999999E+09,8.999999E+09,8.999999E+09,8.999999E+09,8.999999E+09]];
    LOCAL CONST Robtarget Tr_meulage_bavure_12 := [[-109.16,-89.716640625,23],[0.999962143790734,-0.0059959765043272,-0.00628689049226442,0.000484003240229429],[0,0,0,0],[8.999999E+09,8.999999E+09,8.999999E+09,8.999999E+09,8.999999E+09,8.999999E+09]];
    LOCAL CONST Robtarget Tr_meulage_bavure_13 := [[-110.59384375,-88.204296875,23],[0.999962068352189,-0.00604675137594499,-0.00625144268578959,0.000467032071618616],[0,0,0,0],[8.999999E+09,8.999999E+09,8.999999E+09,8.999999E+09,8.999999E+09,8.999999E+09]];
    LOCAL CONST Robtarget Tr_meulage_bavure_14 := [[-113.0693046875,-85.8259921875,23],[0.999962010927491,-0.00608920390131266,-0.00622052361905891,0.000450980709935256],[0,0,0,0],[8.999999E+09,8.999999E+09,8.999999E+09,8.999999E+09,8.999999E+09,8.999999E+09]];
    LOCAL CONST Robtarget Tr_meulage_bavure_15 := [[-116.5336640625,-82.3804765625,23],[0.999961979324864,-0.00612253204756305,-0.00619391853320613,0.000435751340282989],[0,0,0,0],[8.999999E+09,8.999999E+09,8.999999E+09,8.999999E+09,8.999999E+09,8.999999E+09]];
    LOCAL CONST Robtarget Tr_meulage_bavure_16 := [[-120.6395859375,-78.2647890625,23],[0.999961975116599,-0.00614806990931664,-0.00617022512387266,0.000421757302219721],[0,0,0,0],[8.999999E+09,8.999999E+09,8.999999E+09,8.999999E+09,8.999999E+09,8.999999E+09]];
    LOCAL CONST Robtarget Tr_meulage_bavure_17 := [[-123.6929921875,-75.112546875,23],[0.999961994903404,-0.0061689192326601,-0.0061470286788221,0.000408928757118445],[0,0,0,0],[8.999999E+09,8.999999E+09,8.999999E+09,8.999999E+09,8.999999E+09,8.999999E+09]];
    LOCAL CONST Robtarget Tr_meulage_bavure_18 := [[-125.3610546875,-73.3430625,23],[0.999962031172123,-0.00618944812116437,-0.00612119841212377,0.000397336227764191],[0,0,0,0],[8.999999E+09,8.999999E+09,8.999999E+09,8.999999E+09,8.999999E+09,8.999999E+09]];
    LOCAL CONST Robtarget Tr_meulage_bavure_19 := [[-126.754453125,-71.9008203125,23],[0.999962073268793,-0.00621419127235065,-0.00608982978916965,0.000387070983899016],[0,0,0,0],[8.999999E+09,8.999999E+09,8.999999E+09,8.999999E+09,8.999999E+09,8.999999E+09]];
    LOCAL CONST Robtarget Tr_meulage_bavure_20 := [[-127.72003125,-70.9483203125,23],[0.999962110484343,-0.0062463977023955,-0.00605123704480016,0.000377679322043718],[0,0,0,0],[8.999999E+09,8.999999E+09,8.999999E+09,8.999999E+09,8.999999E+09,8.999999E+09]];
    LOCAL CONST Robtarget Tr_meulage_bavure_21 := [[-129.701046875,-68.8303203125,23],[0.999962133219131,-0.00628711119175036,-0.00600565603573082,0.00036939990166719],[0,0,0,0],[8.999999E+09,8.999999E+09,8.999999E+09,8.999999E+09,8.999999E+09,8.999999E+09]];
    LOCAL CONST Robtarget Tr_meulage_bavure_22 := [[-133.266140625,-64.94608984375,23],[0.99996213773405,-0.00633494705063348,-0.00595487565751804,0.000361939383405177],[0,0,0,0],[8.999999E+09,8.999999E+09,8.999999E+09,8.999999E+09,8.999999E+09,8.999999E+09]];
    LOCAL CONST Robtarget Tr_meulage_bavure_23 := [[-136.61690625,-61.2477890625,23],[0.999962126530341,-0.006387099224146,-0.00590122696069222,0.000354948979387185],[0,0,0,0],[8.999999E+09,8.999999E+09,8.999999E+09,8.999999E+09,8.999999E+09,8.999999E+09]];
    LOCAL CONST Robtarget Tr_meulage_bavure_24 := [[-139.611046875,-57.939515625,23],[0.9999621060745,-0.00644106678621852,-0.00584616086352586,0.000348535312339526],[0,0,0,0],[8.999999E+09,8.999999E+09,8.999999E+09,8.999999E+09,8.999999E+09,8.999999E+09]];
    LOCAL CONST Robtarget Tr_meulage_bavure_25 := [[-141.01071875,-56.387984375,23],[0.999962083800876,-0.00649595444071321,-0.00578932566714706,0.000342410328470159],[0,0,0,0],[8.999999E+09,8.999999E+09,8.999999E+09,8.999999E+09,8.999999E+09,8.999999E+09]];
    LOCAL CONST Robtarget Tr_meulage_bavure_26 := [[-142.894984375,-54.19334375,23],[0.999962064519581,-0.00655251804845602,-0.00572894851078868,0.000336419265604524],[0,0,0,0],[8.999999E+09,8.999999E+09,8.999999E+09,8.999999E+09,8.999999E+09,8.999999E+09]];
    LOCAL CONST Robtarget Tr_meulage_bavure_27 := [[-148.83384375,-47.14578125,23],[0.999962048942372,-0.00661208998211344,-0.00566318121263139,0.000330635136995258],[0,0,0,0],[8.999999E+09,8.999999E+09,8.999999E+09,8.999999E+09,8.999999E+09,8.999999E+09]];
    LOCAL CONST Robtarget Tr_meulage_bavure_28 := [[-149.9493125,-45.86146484375,23],[0.999962035831054,-0.00667492806513607,-0.00559167616945523,0.000324637573355],[0,0,0,0],[8.999999E+09,8.999999E+09,8.999999E+09,8.999999E+09,8.999999E+09,8.999999E+09]];
    LOCAL CONST Robtarget Tr_meulage_bavure_29 := [[-150.858,-44.7060234375,23],[0.999962022946597,-0.00673923499407762,-0.00551668136198448,0.000318752245415564],[0,0,0,0],[8.999999E+09,8.999999E+09,8.999999E+09,8.999999E+09,8.999999E+09,8.999999E+09]];
    LOCAL CONST Robtarget Tr_meulage_bavure_30 := [[-152.825828125,-42.34896875,23],[0.999962010172667,-0.00680110908310232,-0.00544290818114873,0.000312853336295676],[0,0,0,0],[8.999999E+09,8.999999E+09,8.999999E+09,8.999999E+09,8.999999E+09,8.999999E+09]];
    LOCAL CONST Robtarget Tr_meulage_bavure_31 := [[-153.0646875,-42.045625,23],[0.999962000082678,-0.00685594733973942,-0.00537589531738725,0.00030680003523034],[0,0,0,0],[8.999999E+09,8.999999E+09,8.999999E+09,8.999999E+09,8.999999E+09,8.999999E+09]];
    LOCAL CONST Robtarget Tr_meulage_bavure_32 := [[-153.298609375,-41.76766796875,23],[0.999961995104879,-0.00690042049080147,-0.00531995900595965,0.000300963611591549],[0,0,0,0],[8.999999E+09,8.999999E+09,8.999999E+09,8.999999E+09,8.999999E+09,8.999999E+09]];
    LOCAL CONST Robtarget Tr_meulage_bavure_33 := [[-155.45503125,-39.067046875,23],[0.999961996654282,-0.00693365037422624,-0.00527661331517334,0.000295112847117237],[0,0,0,0],[8.999999E+09,8.999999E+09,8.999999E+09,8.999999E+09,8.999999E+09,8.999999E+09]];
    LOCAL CONST Robtarget Tr_meulage_bavure_34 := [[-155.83853125,-38.5523359375,23],[0.999962002407522,-0.00695740018143243,-0.00524446395665011,0.00028969235820543],[0,0,0,0],[8.999999E+09,8.999999E+09,8.999999E+09,8.999999E+09,8.999999E+09,8.999999E+09]];
    LOCAL CONST Robtarget Tr_meulage_bavure_35 := [[-159.17671875,-34.22415234375,23],[0.999962007923372,-0.00697524298644607,-0.0052199361139142,0.000284538405505386],[0,0,0,0],[8.999999E+09,8.999999E+09,8.999999E+09,8.999999E+09,8.999999E+09,8.999999E+09]];
    LOCAL CONST Robtarget Tr_meulage_bavure_36 := [[-159.614484375,-33.6722421875,23],[0.999962008667219,-0.006990902201198,-0.00519905462273562,0.000279892235240847],[0,0,0,0],[8.999999E+09,8.999999E+09,8.999999E+09,8.999999E+09,8.999999E+09,8.999999E+09]];
    LOCAL CONST Robtarget Tr_meulage_bavure_37 := [[-164.3065,-27.351958984375,23],[0.999962002263506,-0.00700721250735975,-0.00517849079148398,0.000276107150520898],[0,0,0,0],[8.999999E+09,8.999999E+09,8.999999E+09,8.999999E+09,8.999999E+09,8.999999E+09]];
    LOCAL CONST Robtarget Tr_meulage_bavure_38 := [[-164.679265625,-26.8167109375,23],[0.999961990076073,-0.00702553247341701,-0.00515614194871639,0.000272940962415009],[0,0,0,0],[8.999999E+09,8.999999E+09,8.999999E+09,8.999999E+09,8.999999E+09,8.999999E+09]];
    LOCAL CONST Robtarget Tr_meulage_bavure_39 := [[-165.112953125,-26.228423828125,23],[0.999961975482181,-0.00704590699098499,-0.00513122160660342,0.000270830708944756],[0,0,0,0],[8.999999E+09,8.999999E+09,8.999999E+09,8.999999E+09,8.999999E+09,8.999999E+09]];
    LOCAL CONST Robtarget Tr_meulage_bavure_40 := [[-168.454140625,-21.6435234375,23],[0.999961962412086,-0.00706753358141927,-0.00510400031277217,0.000269960834766814],[0,0,0,0],[8.999999E+09,8.999999E+09,8.999999E+09,8.999999E+09,8.999999E+09,8.999999E+09]];
    LOCAL CONST Robtarget Tr_meulage_bavure_41 := [[-170.152671875,-19.283935546875,23],[0.999961953530477,-0.00708923789455721,-0.00507555615352891,0.000270050586061844],[0,0,0,0],[8.999999E+09,8.999999E+09,8.999999E+09,8.999999E+09,8.999999E+09,8.999999E+09]];
    LOCAL CONST Robtarget Tr_meulage_bavure_42 := [[-170.8105625,-18.345611328125,23],[0.999961949491883,-0.00710998942339345,-0.00504715899000271,0.000271670612758473],[0,0,0,0],[8.999999E+09,8.999999E+09,8.999999E+09,8.999999E+09,8.999999E+09,8.999999E+09]];
    LOCAL CONST Robtarget Tr_meulage_bavure_43 := [[-172.78721875,-15.3552548828125,23],[0.999961952253416,-0.00712897685746209,-0.00501959643461832,0.000274565357887697],[0,0,0,0],[8.999999E+09,8.999999E+09,8.999999E+09,8.999999E+09,8.999999E+09,8.999999E+09]];
    LOCAL CONST Robtarget Tr_meulage_bavure_44 := [[-175.414875,-11.6484072265625,23],[0.999961964220922,-0.0071462207530955,-0.00499238297050297,0.000278841637849669],[0,0,0,0],[8.999999E+09,8.999999E+09,8.999999E+09,8.999999E+09,8.999999E+09,8.999999E+09]];
    LOCAL CONST Robtarget Tr_meulage_bavure_45 := [[-178.3580625,-7.5121767578125,23],[0.999961991280323,-0.00716215131800831,-0.00496372427292004,0.000284648084748537],[0,0,0,0],[8.999999E+09,8.999999E+09,8.999999E+09,8.999999E+09,8.999999E+09,8.999999E+09]];
    LOCAL CONST Robtarget Tr_meulage_bavure_46 := [[-178.55940625,-7.215087890625,23],[0.999962040594633,-0.00717757193983976,-0.00493099574710952,0.000291739280645053],[0,0,0,0],[8.999999E+09,8.999999E+09,8.999999E+09,8.999999E+09,8.999999E+09,8.999999E+09]];
    LOCAL CONST Robtarget Tr_meulage_bavure_47 := [[-178.75059375,-6.9400634765625,23],[0.99996211445084,-0.00719360037323932,-0.00489197779138726,0.000300549436513318],[0,0,0,0],[8.999999E+09,8.999999E+09,8.999999E+09,8.999999E+09,8.999999E+09,8.999999E+09]];
    LOCAL CONST Robtarget Tr_meulage_bavure_48 := [[-180.717390625,-3.98046875,23],[0.999962207543754,-0.00721150559256638,-0.00484573960411499,0.000310610688746849],[0,0,0,0],[8.999999E+09,8.999999E+09,8.999999E+09,8.999999E+09,8.999999E+09,8.999999E+09]];
    LOCAL CONST Robtarget Tr_meulage_bavure_49 := [[-183.206828125,-0.16949462890625,23],[0.999962303541651,-0.00723274614379478,-0.00479323762711521,0.000322105485366172],[0,0,0,0],[8.999999E+09,8.999999E+09,8.999999E+09,8.999999E+09,8.999999E+09,8.999999E+09]];
    LOCAL CONST Robtarget Tr_meulage_bavure_50 := [[-184.33109375,1.59613037109375,23],[0.999962380892266,-0.00725842728211612,-0.00473707579328839,0.000334882948668774],[0,0,0,0],[8.999999E+09,8.999999E+09,8.999999E+09,8.999999E+09,8.999999E+09,8.999999E+09]];
    LOCAL CONST Robtarget Tr_meulage_bavure_51 := [[-185.79925,3.86856079101563,23],[0.999962420961989,-0.00728869412104351,-0.00468080647436497,0.000348787324814613],[0,0,0,0],[8.999999E+09,8.999999E+09,8.999999E+09,8.999999E+09,8.999999E+09,8.999999E+09]];
    LOCAL CONST Robtarget Tr_meulage_bavure_52 := [[-186.629203125,5.2182919921875,23],[0.999962416578377,-0.00732220660990133,-0.0046279914671937,0.00036389019506615],[0,0,0,0],[8.999999E+09,8.999999E+09,8.999999E+09,8.999999E+09,8.999999E+09,8.999999E+09]];
    LOCAL CONST Robtarget Tr_meulage_bavure_53 := [[-188.1745625,7.6268310546875,23],[0.999962375118325,-0.00735623605849889,-0.00458144221385434,0.000380165767094637],[0,0,0,0],[8.999999E+09,8.999999E+09,8.999999E+09,8.999999E+09,8.999999E+09,8.999999E+09]];
    LOCAL CONST Robtarget Tr_meulage_bavure_54 := [[-189.39925,9.66665625,23],[0.999962312722414,-0.00738770291420192,-0.00454278308289721,0.000397620868183864],[0,0,0,0],[8.999999E+09,8.999999E+09,8.999999E+09,8.999999E+09,8.999999E+09,8.999999E+09]];
    LOCAL CONST Robtarget Tr_meulage_bavure_55 := [[-190.449453125,11.194671875,23],[0.999962244973437,-0.00741484182759098,-0.00451171636466311,0.000416129547208],[0,0,0,0],[8.999999E+09,8.999999E+09,8.999999E+09,8.999999E+09,8.999999E+09,8.999999E+09]];
    LOCAL CONST Robtarget Tr_meulage_bavure_56 := [[-193.0021875,15.32894921875,23],[0.999962181220908,-0.00743778642694499,-0.00448616464819334,0.000435646347058839],[0,0,0,0],[8.999999E+09,8.999999E+09,8.999999E+09,8.999999E+09,8.999999E+09,8.999999E+09]];
    LOCAL CONST Robtarget Tr_meulage_bavure_57 := [[-193.809484375,16.6774296875,23],[0.999962122593941,-0.00745867015065665,-0.00446242551786679,0.000456481655128185],[0,0,0,0],[8.999999E+09,8.999999E+09,8.999999E+09,8.999999E+09,8.999999E+09,8.999999E+09]];
    LOCAL CONST Robtarget Tr_meulage_bavure_58 := [[-194.320375,17.45446875,23],[0.999962067884526,-0.00748040563375117,-0.004435926566735,0.000478413159297225],[0,0,0,0],[8.999999E+09,8.999999E+09,8.999999E+09,8.999999E+09,8.999999E+09,8.999999E+09]];
    LOCAL CONST Robtarget Tr_meulage_bavure_59 := [[-197.90896875,23.49331640625,23],[0.999962016551551,-0.00750549685211446,-0.00440244362896079,0.000501459123933804],[0,0,0,0],[8.999999E+09,8.999999E+09,8.999999E+09,8.999999E+09,8.999999E+09,8.999999E+09]];
    LOCAL CONST Robtarget Tr_meulage_bavure_60 := [[-199.941640625,26.863494140625,23],[0.999961971345119,-0.00753479704283086,-0.00435965774700965,0.00052543452096427],[0,0,0,0],[8.999999E+09,8.999999E+09,8.999999E+09,8.999999E+09,8.999999E+09,8.999999E+09]];
    LOCAL CONST Robtarget Tr_meulage_bavure_61 := [[-202.821984375,31.87448046875,23],[0.999961936571014,-0.00756715151347812,-0.00430823922359871,0.000550183525940772],[0,0,0,0],[8.999999E+09,8.999999E+09,8.999999E+09,8.999999E+09,8.999999E+09,8.999999E+09]];
    LOCAL CONST Robtarget Tr_meulage_bavure_62 := [[-203.23153125,32.622771484375,23],[0.999961914008616,-0.00760023964906262,-0.00425150970464612,0.000575807896622991],[0,0,0,0],[8.999999E+09,8.999999E+09,8.999999E+09,8.999999E+09,8.999999E+09,8.999999E+09]];
    LOCAL CONST Robtarget Tr_meulage_bavure_63 := [[-203.5151875,33.11737109375,23],[0.999961907617676,-0.00763080353789807,-0.0041943087189589,0.000601602323278708],[0,0,0,0],[8.999999E+09,8.999999E+09,8.999999E+09,8.999999E+09,8.999999E+09,8.999999E+09]];
    LOCAL CONST Robtarget Tr_meulage_bavure_64 := [[-203.923171875,33.89599609375,23],[0.999961920403614,-0.0076561528400008,-0.00414094644916947,0.000627398527101162],[0,0,0,0],[8.999999E+09,8.999999E+09,8.999999E+09,8.999999E+09,8.999999E+09,8.999999E+09]];
    LOCAL CONST Robtarget Tr_meulage_bavure_65 := [[-208.35253125,42.4410078125,23],[0.99996195726159,-0.00767491084854646,-0.00409309808880888,0.000652932670146597],[0,0,0,0],[8.999999E+09,8.999999E+09,8.999999E+09,8.999999E+09,8.999999E+09,8.999999E+09]];
    LOCAL CONST Robtarget Tr_meulage_bavure_66 := [[-208.638125,42.962890625,23],[0.999962024685903,-0.00768706999961097,-0.00404956459270621,0.000677618993288741],[0,0,0,0],[8.999999E+09,8.999999E+09,8.999999E+09,8.999999E+09,8.999999E+09,8.999999E+09]];
    LOCAL CONST Robtarget Tr_meulage_bavure_67 := [[-209.91159375,45.507203125,23],[0.999962125719391,-0.00769375377706033,-0.00400768852331301,0.000701221986326859],[0,0,0,0],[8.999999E+09,8.999999E+09,8.999999E+09,8.999999E+09,8.999999E+09,8.999999E+09]];
    LOCAL CONST Robtarget Tr_meulage_bavure_68 := [[-211.25371875,48.042296875,23],[0.999962255992443,-0.0076968434545906,-0.00396513647384931,0.00072310724214676],[0,0,0,0],[8.999999E+09,8.999999E+09,8.999999E+09,8.999999E+09,8.999999E+09,8.999999E+09]];
    LOCAL CONST Robtarget Tr_meulage_bavure_69 := [[-211.85778125,49.3566875,23],[0.999962400180486,-0.0076984769342958,-0.00392164294252191,0.000743232672036864],[0,0,0,0],[8.999999E+09,8.999999E+09,8.999999E+09,8.999999E+09,8.999999E+09,8.999999E+09]];
    LOCAL CONST Robtarget Tr_meulage_bavure_70 := [[-212.5911875,50.68365625,23],[0.999962537273801,-0.00770081849109019,-0.00387844343419833,0.000760999367005518],[0,0,0,0],[8.999999E+09,8.999999E+09,8.999999E+09,8.999999E+09,8.999999E+09,8.999999E+09]];
    LOCAL CONST Robtarget Tr_meulage_bavure_71 := [[-214.616,54.92309375,23],[0.999962643796216,-0.00770649390831616,-0.0038364965290926,0.000776052901740392],[0,0,0,0],[8.999999E+09,8.999999E+09,8.999999E+09,8.999999E+09,8.999999E+09,8.999999E+09]];
    LOCAL CONST Robtarget Tr_meulage_bavure_72 := [[-215.722828125,57.05776953125,23],[0.99996270583099,-0.0077178661550509,-0.00379475446098526,0.000788243463504927],[0,0,0,0],[8.999999E+09,8.999999E+09,8.999999E+09,8.999999E+09,8.999999E+09,8.999999E+09]];
    LOCAL CONST Robtarget Tr_meulage_bavure_73 := [[-216.546703125,58.9495234375,23],[0.99996272427158,-0.00773659973320738,-0.00374958041904929,0.000797332183146562],[0,0,0,0],[8.999999E+09,8.999999E+09,8.999999E+09,8.999999E+09,8.999999E+09,8.999999E+09]];
    LOCAL CONST Robtarget Tr_meulage_bavure_74 := [[-217.575921875,60.988984375,23],[0.999962711011017,-0.00776311618167891,-0.00369665048297449,0.000803361595632892],[0,0,0,0],[8.999999E+09,8.999999E+09,8.999999E+09,8.999999E+09,8.999999E+09,8.999999E+09]];
    LOCAL CONST Robtarget Tr_meulage_bavure_75 := [[-218.500390625,63.14721875,23],[0.999962680293283,-0.00779656176933699,-0.00363337877967197,0.000806352214270116],[0,0,0,0],[8.999999E+09,8.999999E+09,8.999999E+09,8.999999E+09,8.999999E+09,8.999999E+09]];
    LOCAL CONST Robtarget Tr_meulage_bavure_76 := [[-220.6359375,68.1213984375,23],[0.999962641539909,-0.00783525413058705,-0.00356011720684244,0.000806153031470366],[0,0,0,0],[8.999999E+09,8.999999E+09,8.999999E+09,8.999999E+09,8.999999E+09,8.999999E+09]];
    LOCAL CONST Robtarget Tr_meulage_bavure_77 := [[-221.501671875,70.223359375,23],[0.999962596694134,-0.00787707091973056,-0.00348030003102254,0.000802793961213237],[0,0,0,0],[8.999999E+09,8.999999E+09,8.999999E+09,8.999999E+09,8.999999E+09,8.999999E+09]];
    LOCAL CONST Robtarget Tr_meulage_bavure_78 := [[-221.745359375,70.870328125,23],[0.999962546346692,-0.00791992353736387,-0.00339799876009892,0.000796441729317385],[0,0,0,0],[8.999999E+09,8.999999E+09,8.999999E+09,8.999999E+09,8.999999E+09,8.999999E+09]];
    LOCAL CONST Robtarget Tr_meulage_bavure_79 := [[-222.486640625,72.465328125,23],[0.999962504672114,-0.00796207510268514,-0.00331281135856404,0.000787331464685115],[0,0,0,0],[8.999999E+09,8.999999E+09,8.999999E+09,8.999999E+09,8.999999E+09,8.999999E+09]];
    LOCAL CONST Robtarget Tr_meulage_bavure_80 := [[-222.990421875,73.6807890625,23],[0.999962504866291,-0.00800218934101718,-0.0032175098712562,0.000775536918636133],[0,0,0,0],[8.999999E+09,8.999999E+09,8.999999E+09,8.999999E+09,8.999999E+09,8.999999E+09]];
    LOCAL CONST Robtarget Tr_meulage_bavure_81 := [[-224.275796875,76.966890625,23],[0.999962608577845,-0.00803941635276192,-0.00309356502406099,0.00076097722688008],[0,0,0,0],[8.999999E+09,8.999999E+09,8.999999E+09,8.999999E+09,8.999999E+09,8.999999E+09]];
    LOCAL CONST Robtarget Tr_meulage_bavure_82 := [[-225.08675,78.7561640625,23],[0.999962886200099,-0.00807428344837244,-0.00291170692716225,0.000744400385413021],[0,0,0,0],[8.999999E+09,8.999999E+09,8.999999E+09,8.999999E+09,8.999999E+09,8.999999E+09]];
    LOCAL CONST Robtarget Tr_meulage_bavure_83 := [[-225.64590625,79.798890625,23],[0.999963392677705,-0.00810739824897129,-0.00263753787119351,0.000725804453396599],[0,0,0,0],[8.999999E+09,8.999999E+09,8.999999E+09,8.999999E+09,8.999999E+09,8.999999E+09]];
    LOCAL CONST Robtarget Tr_meulage_bavure_84 := [[-225.846171875,80.3101484375,23],[0.99996415909543,-0.00813468420304933,-0.00223818202998894,0.000705676049909828],[0,0,0,0],[8.999999E+09,8.999999E+09,8.999999E+09,8.999999E+09,8.999999E+09,8.999999E+09]];
    LOCAL CONST Robtarget Tr_meulage_bavure_85 := [[-227.168125,83.241515625,23],[0.999965163296161,-0.0081443667192934,-0.00169510125001401,0.00068419045335726],[0,0,0,0],[8.999999E+09,8.999999E+09,8.999999E+09,8.999999E+09,8.999999E+09,8.999999E+09]];
    LOCAL CONST Robtarget Tr_meulage_bavure_86 := [[-227.25865625,83.4700625,23],[0.999966372018882,-0.00811202168150841,-0.00100627109284766,0.000661327543930723],[0,0,0,0],[8.999999E+09,8.999999E+09,8.999999E+09,8.999999E+09,8.999999E+09,8.999999E+09]];
    LOCAL CONST Robtarget Tr_meulage_bavure_87 := [[-227.48228125,84.181734375,23],[0.999967778293875,-0.00800020643552291,-0.000183585603731339,0.000636684636958335],[0,0,0,0],[8.999999E+09,8.999999E+09,8.999999E+09,8.999999E+09,8.999999E+09,8.999999E+09]];
    LOCAL CONST Robtarget Tr_meulage_bavure_88 := [[-228.1584375,86.6586875,23],[0.99996936369207,-0.00776739897477166,0.000753168095225507,0.000609859216494483],[0,0,0,0],[8.999999E+09,8.999999E+09,8.999999E+09,8.999999E+09,8.999999E+09,8.999999E+09]];
    LOCAL CONST Robtarget Tr_meulage_bavure_89 := [[-227.72525,89.4899609375,23],[0.999970990002363,-0.00738303481384577,0.00178132270621163,0.000580379226996989],[0,0,0,0],[8.999999E+09,8.999999E+09,8.999999E+09,8.999999E+09,8.999999E+09,8.999999E+09]];
    LOCAL CONST Robtarget Tr_meulage_bavure_90 := [[-227.624265625,89.8831484375,23],[0.999972304282206,-0.006844928157311,0.0028702030807366,0.000547321962850733],[0,0,0,0],[8.999999E+09,8.999999E+09,8.999999E+09,8.999999E+09,8.999999E+09,8.999999E+09]];
    LOCAL CONST Robtarget Tr_meulage_bavure_91 := [[-226.95615625,90.7658046875,23],[0.999972826610504,-0.00618791908953869,0.00397436400981398,0.000510028094337078],[0,0,0,0],[8.999999E+09,8.999999E+09,8.999999E+09,8.999999E+09,8.999999E+09,8.999999E+09]];
    LOCAL CONST Robtarget Tr_meulage_bavure_92 := [[-226.279703125,91.630984375,23],[0.999972218417723,-0.00547963547171994,0.00503160099910544,0.00046795215622161],[0,0,0,0],[8.999999E+09,8.999999E+09,8.999999E+09,8.999999E+09,8.999999E+09,8.999999E+09]];
    LOCAL CONST Robtarget Tr_meulage_bavure_93 := [[-223.598421875,93.2830234375,23],[0.99997054999118,-0.00480121039563465,0.00597244441723303,0.000421232426433095],[0,0,0,0],[8.999999E+09,8.999999E+09,8.999999E+09,8.999999E+09,8.999999E+09,8.999999E+09]];
    LOCAL CONST Robtarget Tr_meulage_bavure_94 := [[-223.413234375,93.4259609375,23],[0.999968299201887,-0.00422185887336958,0.00674084915521702,0.000370744663549541],[0,0,0,0],[8.999999E+09,8.999999E+09,8.999999E+09,8.999999E+09,8.999999E+09,8.999999E+09]];
    LOCAL CONST Robtarget Tr_meulage_bavure_95 := [[-222.693234375,93.70434375,23],[0.999966079084191,-0.00378045450501961,0.00731083217890477,0.000317139682157139],[0,0,0,0],[8.999999E+09,8.999999E+09,8.999999E+09,8.999999E+09,8.999999E+09,8.999999E+09]];
    LOCAL CONST Robtarget Tr_meulage_bavure_96 := [[-219.287515625,94.9596875,23],[0.999964327519385,-0.00348177564855813,0.00769108597345516,0.000261004954059566],[0,0,0,0],[8.999999E+09,8.999999E+09,8.999999E+09,8.999999E+09,8.999999E+09,8.999999E+09]];
    LOCAL CONST Robtarget Tr_meulage_bavure_97 := [[-215.06440625,96.426359375,23],[0.999963170875546,-0.00330407640619514,0.00791825498578845,0.000203001489913422],[0,0,0,0],[8.999999E+09,8.999999E+09,8.999999E+09,8.999999E+09,8.999999E+09,8.999999E+09]];
    LOCAL CONST Robtarget Tr_meulage_bavure_98 := [[-207.5475,99.17565625,23],[0.999962519546413,-0.00321413343811005,0.00803793058954246,0.000143249675280452],[0,0,0,0],[8.999999E+09,8.999999E+09,8.999999E+09,8.999999E+09,8.999999E+09,8.999999E+09]];
    LOCAL CONST Robtarget Tr_meulage_bavure_99 := [[-202.719625,100.9839765625,23],[0.999962198739105,-0.00317882241630533,0.00809255806703144,8.1760817975787E-05],[0,0,0,0],[8.999999E+09,8.999999E+09,8.999999E+09,8.999999E+09,8.999999E+09,8.999999E+09]];
    LOCAL CONST Robtarget Tr_meulage_bavure_100 := [[-200.20753125,101.9860859375,23],[0.999962057510683,-0.00317230715018142,0.00811293167414166,1.86010235049611E-05],[0,0,0,0],[8.999999E+09,8.999999E+09,8.999999E+09,8.999999E+09,8.999999E+09,8.999999E+09]];
    LOCAL CONST Robtarget Tr_meulage_bavure_101 := [[-192.306046875,105.0720859375,23],[0.999962002712386,-0.00317681158588654,0.0081178138815739,-4.57970189765234E-05],[0,0,0,0],[8.999999E+09,8.999999E+09,8.999999E+09,8.999999E+09,8.999999E+09,8.999999E+09]];
    LOCAL CONST Robtarget Tr_meulage_bavure_102 := [[-188.0050625,106.8087734375,23],[0.999961980266291,-0.00318078388931623,0.00811839058369918,-0.000111220941386237],[0,0,0,0],[8.999999E+09,8.999999E+09,8.999999E+09,8.999999E+09,8.999999E+09,8.999999E+09]];
    LOCAL CONST Robtarget Tr_meulage_bavure_103 := [[-184.288375,108.2283046875,23],[0.999961972184813,-0.00318004150486139,0.00811849290295125,-0.00017774496020173],[0,0,0,0],[8.999999E+09,8.999999E+09,8.999999E+09,8.999999E+09,8.999999E+09,8.999999E+09]];
    LOCAL CONST Robtarget Tr_meulage_bavure_104 := [[-182.750859375,108.85690625,23],[0.999961971302312,-0.00317464804029052,0.008118968891496,-0.000244751207947974],[0,0,0,0],[8.999999E+09,8.999999E+09,8.999999E+09,8.999999E+09,8.999999E+09,8.999999E+09]];
    LOCAL CONST Robtarget Tr_meulage_bavure_105 := [[-175.827140625,111.3243125,23],[0.999961975157325,-0.00316737815884235,0.00811904307818454,-0.000311599993234516],[0,0,0,0],[8.999999E+09,8.999999E+09,8.999999E+09,8.999999E+09,8.999999E+09,8.999999E+09]];
    LOCAL CONST Robtarget Tr_meulage_bavure_106 := [[-173.832390625,112.04565625,23],[0.99996198617059,-0.00316137549150996,0.00811720406612392,-0.000378043542401515],[0,0,0,0],[8.999999E+09,8.999999E+09,8.999999E+09,8.999999E+09,8.999999E+09,8.999999E+09]];
    LOCAL CONST Robtarget Tr_meulage_bavure_107 := [[-173.1296875,112.2573515625,23],[0.999962006836233,-0.00315701494634037,0.0081130440976403,-0.000443459300507456],[0,0,0,0],[8.999999E+09,8.999999E+09,8.999999E+09,8.999999E+09,8.999999E+09,8.999999E+09]];
    LOCAL CONST Robtarget Tr_meulage_bavure_108 := [[-172.613578125,112.4072578125,23],[0.999962038359955,-0.00315154488546206,0.00810755522228131,-0.000507101722911426],[0,0,0,0],[8.999999E+09,8.999999E+09,8.999999E+09,8.999999E+09,8.999999E+09,8.999999E+09]];
    LOCAL CONST Robtarget Tr_meulage_bavure_109 := [[-171.29321875,112.818390625,23],[0.999962079788997,-0.00314043242189349,0.00810269302694749,-0.000568360781350699],[0,0,0,0],[8.999999E+09,8.999999E+09,8.999999E+09,8.999999E+09,8.999999E+09,8.999999E+09]];
    LOCAL CONST Robtarget Tr_meulage_bavure_110 := [[-166.94565625,114.5949375,23],[0.999962127822257,-0.00312047030854098,0.00810017544485492,-0.000626692906809977],[0,0,0,0],[8.999999E+09,8.999999E+09,8.999999E+09,8.999999E+09,8.999999E+09,8.999999E+09]];
    LOCAL CONST Robtarget Tr_meulage_bavure_111 := [[-166.10790625,114.9887421875,23],[0.999962177741736,-0.00309308021074327,0.00810012041765288,-0.000681168139952983],[0,0,0,0],[8.999999E+09,8.999999E+09,8.999999E+09,8.999999E+09,8.999999E+09,8.999999E+09]];
    LOCAL CONST Robtarget Tr_meulage_bavure_112 := [[-165.576859375,115.1702890625,23],[0.999962227620716,-0.00306456086880033,0.00810045070758978,-0.000731092901727558],[0,0,0,0],[8.999999E+09,8.999999E+09,8.999999E+09,8.999999E+09,8.999999E+09,8.999999E+09]];
    LOCAL CONST Robtarget Tr_meulage_bavure_113 := [[-156.145875,118.6306171875,23],[0.999962283412205,-0.00304461906697268,0.00809694449541714,-0.000775588566238419],[0,0,0,0],[8.999999E+09,8.999999E+09,8.999999E+09,8.999999E+09,8.999999E+09,8.999999E+09]];
    LOCAL CONST Robtarget Tr_meulage_bavure_114 := [[-154.747203125,119.1098359375,23],[0.999962357808097,-0.00304265457332692,0.00808469096427415,-0.000814243225873381],[0,0,0,0],[8.999999E+09,8.999999E+09,8.999999E+09,8.999999E+09,8.999999E+09,8.999999E+09]];
    LOCAL CONST Robtarget Tr_meulage_bavure_115 := [[-152.75003125,119.97128125,23],[0.99996246450818,-0.00306424450113968,0.00805999899799525,-0.000846402100787465],[0,0,0,0],[8.999999E+09,8.999999E+09,8.999999E+09,8.999999E+09,8.999999E+09,8.999999E+09]];
    LOCAL CONST Robtarget Tr_meulage_bavure_116 := [[-150.449125,120.91678125,23],[0.99996260556245,-0.00310923364557221,0.00802246661457766,-0.000871878610622737],[0,0,0,0],[8.999999E+09,8.999999E+09,8.999999E+09,8.999999E+09,8.999999E+09,8.999999E+09]];
    LOCAL CONST Robtarget Tr_meulage_bavure_117 := [[-147.3660625,122.18359375,23],[0.999962764428348,-0.00317146905849651,0.00797612270791459,-0.00089050961580384],[0,0,0,0],[8.999999E+09,8.999999E+09,8.999999E+09,8.999999E+09,8.999999E+09,8.999999E+09]];
    LOCAL CONST Robtarget Tr_meulage_bavure_118 := [[-143.346625,123.634,23],[0.999962907595264,-0.00324109376905866,0.00792870666539526,-0.000902416433717018],[0,0,0,0],[8.999999E+09,8.999999E+09,8.999999E+09,8.999999E+09,8.999999E+09,8.999999E+09]];
    LOCAL CONST Robtarget Tr_meulage_bavure_119 := [[-139.0588125,125.2717578125,23],[0.999962996851252,-0.00330716884475989,0.00788945117244093,-0.000907812036375465],[0,0,0,0],[8.999999E+09,8.999999E+09,8.999999E+09,8.999999E+09,8.999999E+09,8.999999E+09]];
    LOCAL CONST Robtarget Tr_meulage_bavure_120 := [[-138.84503125,125.374359375,23],[0.999963004540385,-0.00336124660347364,0.00786561265263907,-0.000907584395994368],[0,0,0,0],[8.999999E+09,8.999999E+09,8.999999E+09,8.999999E+09,8.999999E+09,8.999999E+09]];
    LOCAL CONST Robtarget Tr_meulage_bavure_121 := [[-138.535,125.5080234375,23],[0.999962924579735,-0.00339984446327613,0.0078597937812037,-0.000902311080516937],[0,0,0,0],[8.999999E+09,8.999999E+09,8.999999E+09,8.999999E+09,8.999999E+09,8.999999E+09]];
    LOCAL CONST Robtarget Tr_meulage_bavure_122 := [[-130.47903125,128.7274765625,23],[0.999962773093055,-0.00342468685382083,0.00786934735934486,-0.000892927846553077],[0,0,0,0],[8.999999E+09,8.999999E+09,8.999999E+09,8.999999E+09,8.999999E+09,8.999999E+09]];
    LOCAL CONST Robtarget Tr_meulage_bavure_123 := [[-129.8134453125,129.150546875,23],[0.99996258056934,-0.00344169753573675,0.00788777136981549,-0.00088047827728923],[0,0,0,0],[8.999999E+09,8.999999E+09,8.999999E+09,8.999999E+09,8.999999E+09,8.999999E+09]];
    LOCAL CONST Robtarget Tr_meulage_bavure_124 := [[-129.0030234375,129.4828828125,23],[0.999962380294223,-0.00345731776111768,0.00790788510354003,-0.000866200553298891],[0,0,0,0],[8.999999E+09,8.999999E+09,8.999999E+09,8.999999E+09,8.999999E+09,8.999999E+09]];
    LOCAL CONST Robtarget Tr_meulage_bavure_125 := [[-126.592984375,130.564484375,23],[0.99996219785947,-0.00347561839350825,0.00792449965678643,-0.000851606734328924],[0,0,0,0],[8.999999E+09,8.999999E+09,8.999999E+09,8.999999E+09,8.999999E+09,8.999999E+09]];
    LOCAL CONST Robtarget Tr_meulage_bavure_126 := [[-124.177125,131.57909375,23],[0.999962047414002,-0.00349717696839534,0.00793544718678285,-0.000837951546620016],[0,0,0,0],[8.999999E+09,8.999999E+09,8.999999E+09,8.999999E+09,8.999999E+09,8.999999E+09]];
    LOCAL CONST Robtarget Tr_meulage_bavure_127 := [[-119.71090625,133.578453125,23],[0.999961932565298,-0.00351939049529787,0.00794130438487171,-0.000826435408230126],[0,0,0,0],[8.999999E+09,8.999999E+09,8.999999E+09,8.999999E+09,8.999999E+09,8.999999E+09]];
    LOCAL CONST Robtarget Tr_meulage_bavure_128 := [[-115.9326171875,134.801296875,23],[0.99996185176171,-0.00353841375766718,0.00794386902647688,-0.000818287395994475],[0,0,0,0],[8.999999E+09,8.999999E+09,8.999999E+09,8.999999E+09,8.999999E+09,8.999999E+09]];
    LOCAL CONST Robtarget Tr_meulage_bavure_129 := [[-112.962375,136.22165625,23],[0.999961804385776,-0.00354860887609422,0.00794566822002104,-0.000814555783895983],[0,0,0,0],[8.999999E+09,8.999999E+09,8.999999E+09,8.999999E+09,8.999999E+09,8.999999E+09]];
    LOCAL CONST Robtarget Tr_meulage_bavure_130 := [[-108.40240625,137.73059375,23],[0.999961792053304,-0.00354353053329675,0.00794934563034343,-0.000815922149177589],[0,0,0,0],[8.999999E+09,8.999999E+09,8.999999E+09,8.999999E+09,8.999999E+09,8.999999E+09]];
    LOCAL CONST Robtarget Tr_meulage_bavure_131 := [[-108.1422109375,137.8111875,23],[0.999961820984418,-0.00351453147262193,0.00795787932797097,-0.000822677735411536],[0,0,0,0],[8.999999E+09,8.999999E+09,8.999999E+09,8.999999E+09,8.999999E+09,8.999999E+09]];
    LOCAL CONST Robtarget Tr_meulage_bavure_132 := [[-107.3793359375,138.154171875,23],[0.999961896374584,-0.00345318062695781,0.00797395328200829,-0.000835111705077773],[0,0,0,0],[8.999999E+09,8.999999E+09,8.999999E+09,8.999999E+09,8.999999E+09,8.999999E+09]];
    LOCAL CONST Robtarget Tr_meulage_bavure_133 := [[-104.032625,139.779359375,23],[0.999962020186661,-0.00335637675049039,0.00799785392570132,-0.000852790656710937],[0,0,0,0],[8.999999E+09,8.999999E+09,8.999999E+09,8.999999E+09,8.999999E+09,8.999999E+09]];
    LOCAL CONST Robtarget Tr_meulage_bavure_134 := [[-103.578125,139.663328125,23],[0.999962188433737,-0.00323099950134897,0.00802602397659707,-0.000874805213175378],[0,0,0,0],[8.999999E+09,8.999999E+09,8.999999E+09,8.999999E+09,8.999999E+09,8.999999E+09]];
    LOCAL CONST Robtarget Tr_meulage_bavure_135 := [[-98.273375,140.78409375,23],[0.999962399097285,-0.00309571010177302,0.00805024654358526,-0.000900278376305992],[0,0,0,0],[8.999999E+09,8.999999E+09,8.999999E+09,8.999999E+09,8.999999E+09,8.999999E+09]];
    LOCAL CONST Robtarget Tr_meulage_bavure_136 := [[-94.0906640625,142.32440625,23],[0.999962668410932,-0.00297502914782558,0.00805919384918282,-0.000927567010956075],[0,0,0,0],[8.999999E+09,8.999999E+09,8.999999E+09,8.999999E+09,8.999999E+09,8.999999E+09]];
    LOCAL CONST Robtarget Tr_meulage_bavure_137 := [[-90.7126171875,142.525,23],[0.999963027352481,-0.00289318362611431,0.00804121796472182,-0.000955107433916964],[0,0,0,0],[8.999999E+09,8.999999E+09,8.999999E+09,8.999999E+09,8.999999E+09,8.999999E+09]];
    LOCAL CONST Robtarget Tr_meulage_bavure_138 := [[-86.2345,143.279234375,23],[0.99996350480306,-0.00286763554286156,0.00798765868892909,-0.000981344507649053],[0,0,0,0],[8.999999E+09,8.999999E+09,8.999999E+09,8.999999E+09,8.999999E+09,8.999999E+09]];
    LOCAL CONST Robtarget Tr_meulage_bavure_139 := [[-86.203125,143.292453125,23],[0.999964101004759,-0.00290835054051546,0.00789488200155513,-0.0010045083663982],[0,0,0,0],[8.999999E+09,8.999999E+09,8.999999E+09,8.999999E+09,8.999999E+09,8.999999E+09]];
    LOCAL CONST Robtarget Tr_meulage_bavure_140 := [[-82.192140625,145.729125,23],[0.999964765007298,-0.00301961993185755,0.00776556585570944,-0.00102304755877],[0,0,0,0],[8.999999E+09,8.999999E+09,8.999999E+09,8.999999E+09,8.999999E+09,8.999999E+09]];
    LOCAL CONST Robtarget Tr_meulage_bavure_141 := [[-78.507078125,145.4126875,23],[0.999965393633565,-0.00320114174655763,0.00760864225451013,-0.00103575568100327],[0,0,0,0],[8.999999E+09,8.999999E+09,8.999999E+09,8.999999E+09,8.999999E+09,8.999999E+09]];
    LOCAL CONST Robtarget Tr_meulage_bavure_142 := [[-75.921390625,146.10934375,23],[0.999965854042376,-0.00344174621643286,0.00744044368221778,-0.00104159977682935],[0,0,0,0],[8.999999E+09,8.999999E+09,8.999999E+09,8.999999E+09,8.999999E+09,8.999999E+09]];
    LOCAL CONST Robtarget Tr_meulage_bavure_143 := [[-74.7984609375,147.043796875,23],[0.999966033387402,-0.00371257439493688,0.0072847327268195,-0.00103996727140966],[0,0,0,0],[8.999999E+09,8.999999E+09,8.999999E+09,8.999999E+09,8.999999E+09,8.999999E+09]];
    LOCAL CONST Robtarget Tr_meulage_bavure_144 := [[-73.9298984375,147.591828125,23],[0.999965901664432,-0.00396580155588741,0.00716979073944989,-0.00103054704499335],[0,0,0,0],[8.999999E+09,8.999999E+09,8.999999E+09,8.999999E+09,8.999999E+09,8.999999E+09]];
    LOCAL CONST Robtarget Tr_meulage_bavure_145 := [[-67.570890625,150.951265625,23],[0.999965530320044,-0.0041456594635002,0.00712210369143447,-0.00101356715334612],[0,0,0,0],[8.999999E+09,8.999999E+09,8.999999E+09,8.999999E+09,8.999999E+09,8.999999E+09]];
    LOCAL CONST Robtarget Tr_meulage_bavure_146 := [[-66.9260546875,151.566953125,23],[0.999965045741767,-0.00420781759119842,0.00715698973872769,-0.000989476460184934],[0,0,0,0],[8.999999E+09,8.999999E+09,8.999999E+09,8.999999E+09,8.999999E+09,8.999999E+09]];
    LOCAL CONST Robtarget Tr_meulage_bavure_147 := [[-64.8245859375,153.340125,23],[0.999964541045771,-0.00413745962110207,0.00727175503878185,-0.000958987831283091],[0,0,0,0],[8.999999E+09,8.999999E+09,8.999999E+09,8.999999E+09,8.999999E+09,8.999999E+09]];
    LOCAL CONST Robtarget Tr_meulage_bavure_148 := [[-62.8503125,154.698546875,23],[0.999964033470352,-0.00395785794312318,0.00744415070581602,-0.000922901119298366],[0,0,0,0],[8.999999E+09,8.999999E+09,8.999999E+09,8.999999E+09,8.999999E+09,8.999999E+09]];
    LOCAL CONST Robtarget Tr_meulage_bavure_149 := [[-62.48559375,154.97553125,23],[0.999963511950311,-0.00371876726770496,0.00763985236910044,-0.000882152927775635],[0,0,0,0],[8.999999E+09,8.999999E+09,8.999999E+09,8.999999E+09,8.999999E+09,8.999999E+09]];
    LOCAL CONST Robtarget Tr_meulage_bavure_150 := [[-59.9157109375,155.998328125,23],[0.999962995516677,-0.00347726400481399,0.00782398627675476,-0.000837538713477078],[0,0,0,0],[8.999999E+09,8.999999E+09,8.999999E+09,8.999999E+09,8.999999E+09,8.999999E+09]];
    LOCAL CONST Robtarget Tr_meulage_bavure_151 := [[-58.8825703125,156.425390625,23],[0.999962541733171,-0.00327702862620634,0.00797196873925292,-0.000789891346532901],[0,0,0,0],[8.999999E+09,8.999999E+09,8.999999E+09,8.999999E+09,8.999999E+09,8.999999E+09]];
    LOCAL CONST Robtarget Tr_meulage_bavure_152 := [[-56.307375,157.295984375,23],[0.999962202903579,-0.00313880610895622,0.00807417553490213,-0.000740506490670864],[0,0,0,0],[8.999999E+09,8.999999E+09,8.999999E+09,8.999999E+09,8.999999E+09,8.999999E+09]];
    LOCAL CONST Robtarget Tr_meulage_bavure_153 := [[-52.86923046875,158.493984375,23],[0.999961992313195,-0.0030613597451768,0.00813421517442683,-0.000690325309601794],[0,0,0,0],[8.999999E+09,8.999999E+09,8.999999E+09,8.999999E+09,8.999999E+09,8.999999E+09]];
    LOCAL CONST Robtarget Tr_meulage_bavure_154 := [[-51.7835703125,158.931546875,23],[0.99996188741909,-0.0030299724563962,0.00816290360829594,-0.000640297466473176],[0,0,0,0],[8.999999E+09,8.999999E+09,8.999999E+09,8.999999E+09,8.999999E+09,8.999999E+09]];
    LOCAL CONST Robtarget Tr_meulage_bavure_155 := [[-40.98583984375,163.068,23],[0.999961850890602,-0.00302700638485328,0.0081721516004211,-0.000591552201330631],[0,0,0,0],[8.999999E+09,8.999999E+09,8.999999E+09,8.999999E+09,8.999999E+09,8.999999E+09]];
    LOCAL CONST Robtarget Tr_meulage_bavure_156 := [[-38.021515625,164.108671875,23],[0.99996185114879,-0.00303731555997685,0.00817155844881757,-0.000544604252895512],[0,0,0,0],[8.999999E+09,8.999999E+09,8.999999E+09,8.999999E+09,8.999999E+09,8.999999E+09]];
    LOCAL CONST Robtarget Tr_meulage_bavure_157 := [[-35.14184375,165.060328125,23],[0.999961868394205,-0.00305062007744611,0.00816734053037751,-0.000500023373652828],[0,0,0,0],[8.999999E+09,8.999999E+09,8.999999E+09,8.999999E+09,8.999999E+09,8.999999E+09]];
    LOCAL CONST Robtarget Tr_meulage_bavure_158 := [[-33.10540625,165.86828125,23],[0.999961891207317,-0.00306066157509411,0.00816324375551864,-0.000458186858916613],[0,0,0,0],[8.999999E+09,8.999999E+09,8.999999E+09,8.999999E+09,8.999999E+09,8.999999E+09]];
    LOCAL CONST Robtarget Tr_meulage_bavure_159 := [[-27.68307421875,168.024234375,23],[0.999961915392948,-0.0030649271371925,0.00816079138274002,-0.00041889057874854],[0,0,0,0],[8.999999E+09,8.999999E+09,8.999999E+09,8.999999E+09,8.999999E+09,8.999999E+09]];
    LOCAL CONST Robtarget Tr_meulage_bavure_160 := [[-25.93048046875,168.741875,23],[0.999961938775197,-0.00306389068063115,0.00816011465737349,-0.000382235039404185],[0,0,0,0],[8.999999E+09,8.999999E+09,8.999999E+09,8.999999E+09,8.999999E+09,8.999999E+09]];
    LOCAL CONST Robtarget Tr_meulage_bavure_161 := [[-23.64306640625,169.603484375,23],[0.999961960302185,-0.00306012324054547,0.00816042469411037,-0.00034794134108323],[0,0,0,0],[8.999999E+09,8.999999E+09,8.999999E+09,8.999999E+09,8.999999E+09,8.999999E+09]];
    LOCAL CONST Robtarget Tr_meulage_bavure_162 := [[-21.365294921875,170.37096875,23],[0.999961979735883,-0.00305747395378072,0.00816035173325937,-0.000315587239850761],[0,0,0,0],[8.999999E+09,8.999999E+09,8.999999E+09,8.999999E+09,8.999999E+09,8.999999E+09]];
    LOCAL CONST Robtarget Tr_meulage_bavure_163 := [[-16.819091796875,171.9710625,23],[0.999961996429122,-0.00305940427325669,0.00815871585136572,-0.00028477821974555],[0,0,0,0],[8.999999E+09,8.999999E+09,8.999999E+09,8.999999E+09,8.999999E+09,8.999999E+09]];
    LOCAL CONST Robtarget Tr_meulage_bavure_164 := [[-15.8587646484375,172.287046875,23],[0.999962009082445,-0.00306753312488859,0.00815508639927683,-0.000255339280834352],[0,0,0,0],[8.999999E+09,8.999999E+09,8.999999E+09,8.999999E+09,8.999999E+09,8.999999E+09]];
    LOCAL CONST Robtarget Tr_meulage_bavure_165 := [[-12.4654541015625,173.585234375,23],[0.999962016304588,-0.00308116498904918,0.00814989918196505,-0.000226966290859731],[0,0,0,0],[8.999999E+09,8.999999E+09,8.999999E+09,8.999999E+09,8.999999E+09,8.999999E+09]];
    LOCAL CONST Robtarget Tr_meulage_bavure_166 := [[-5.41607666015625,176.28353125,23],[0.999962017223252,-0.00309772161053187,0.0081442300207079,-0.000199371508450525],[0,0,0,0],[8.999999E+09,8.999999E+09,8.999999E+09,8.999999E+09,8.999999E+09,8.999999E+09]];
    LOCAL CONST Robtarget Tr_meulage_bavure_167 := [[-0.180450439453125,178.310421875,23],[0.999962012189987,-0.00311410975184325,0.00813921386831294,-0.000172322407015176],[0,0,0,0],[8.999999E+09,8.999999E+09,8.999999E+09,8.999999E+09,8.999999E+09,8.999999E+09]];
    LOCAL CONST Robtarget Tr_meulage_bavure_168 := [[1.27627563476563,178.891109375,23],[0.999962002813457,-0.0031279825450031,0.0081355625664491,-0.000145863721368929],[0,0,0,0],[8.999999E+09,8.999999E+09,8.999999E+09,8.999999E+09,8.999999E+09,8.999999E+09]];
    LOCAL CONST Robtarget Tr_meulage_bavure_169 := [[5.4862978515625,180.55865625,23],[0.999961991512202,-0.00313822044893878,0.00813343248110741,-0.000119914300107874],[0,0,0,0],[8.999999E+09,8.999999E+09,8.999999E+09,8.999999E+09,8.999999E+09,8.999999E+09]];
    LOCAL CONST Robtarget Tr_meulage_bavure_170 := [[9.74334765625,182.21846875,23],[0.999961980594123,-0.00314482968136967,0.00813255547720585,-9.46253826712253E-05],[0,0,0,0],[8.999999E+09,8.999999E+09,8.999999E+09,8.999999E+09,8.999999E+09,8.999999E+09]];
    LOCAL CONST Robtarget Tr_meulage_bavure_171 := [[15.357849609375,184.33625,23],[0.999961971894974,-0.00314798370694139,0.00813265563153133,-6.98203021213653E-05],[0,0,0,0],[8.999999E+09,8.999999E+09,8.999999E+09,8.999999E+09,8.999999E+09,8.999999E+09]];
    LOCAL CONST Robtarget Tr_meulage_bavure_172 := [[18.40124609375,185.537328125,23],[0.999961966534095,-0.00314699463706648,0.00813386894060149,-4.56736016241858E-05],[0,0,0,0],[8.999999E+09,8.999999E+09,8.999999E+09,8.999999E+09,8.999999E+09,8.999999E+09]];
    LOCAL CONST Robtarget Tr_meulage_bavure_173 := [[22.57159375,187.19659375,23],[0.999961964936754,-0.00314039586678054,0.00813671293343103,-2.22769846104202E-05],[0,0,0,0],[8.999999E+09,8.999999E+09,8.999999E+09,8.999999E+09,8.999999E+09,8.999999E+09]];
    LOCAL CONST Robtarget Tr_meulage_bavure_174 := [[22.874939453125,187.317625,23],[0.999961966541119,-0.00312727232604969,0.00814159928766936,2.36617836002376E-07],[0,0,0,0],[8.999999E+09,8.999999E+09,8.999999E+09,8.999999E+09,8.999999E+09,8.999999E+09]];
    LOCAL CONST Robtarget Tr_meulage_bavure_175 := [[23.29376171875,187.488734375,23],[0.999961969815532,-0.00310880343220283,0.00814823829406786,2.18303410683885E-05],[0,0,0,0],[8.999999E+09,8.999999E+09,8.999999E+09,8.999999E+09,8.999999E+09,8.999999E+09]];
    LOCAL CONST Robtarget Tr_meulage_bavure_176 := [[32.046173828125,191.0809375,23],[0.999961972768327,-0.00308907254819846,0.00815529582547703,4.24036205965828E-05],[0,0,0,0],[8.999999E+09,8.999999E+09,8.999999E+09,8.999999E+09,8.999999E+09,8.999999E+09]];
    LOCAL CONST Robtarget Tr_meulage_bavure_177 := [[37.37878515625,193.0600625,23],[0.999961973659064,-0.00307447853060614,0.00816057457920139,6.19691152862939E-05],[0,0,0,0],[8.999999E+09,8.999999E+09,8.999999E+09,8.999999E+09,8.999999E+09,8.999999E+09]];
    LOCAL CONST Robtarget Tr_meulage_bavure_178 := [[37.698578125,193.17725,23],[0.999961975251196,-0.00307059042721957,0.00816168127780856,8.05287221932766E-05],[0,0,0,0],[8.999999E+09,8.999999E+09,8.999999E+09,8.999999E+09,8.999999E+09,8.999999E+09]];
    LOCAL CONST Robtarget Tr_meulage_bavure_179 := [[40.8884296875,194.392734375,23],[0.999961984568465,-0.00307948056879309,0.00815699639541662,9.81179283847894E-05],[0,0,0,0],[8.999999E+09,8.999999E+09,8.999999E+09,8.999999E+09,8.999999E+09,8.999999E+09]];
    LOCAL CONST Robtarget Tr_meulage_bavure_180 := [[45.28210546875,196.084015625,23],[0.999962015801729,-0.00309709486986929,0.00814627596830792,0.000114651463663724],[0,0,0,0],[8.999999E+09,8.999999E+09,8.999999E+09,8.999999E+09,8.999999E+09,8.999999E+09]];
    LOCAL CONST Robtarget Tr_meulage_bavure_181 := [[49.8389296875,197.72396875,23],[0.999962107062313,-0.00310872382553934,0.00813039921741304,0.00012993937861946],[0,0,0,0],[8.999999E+09,8.999999E+09,8.999999E+09,8.999999E+09,8.999999E+09,8.999999E+09]];
    LOCAL CONST Robtarget Tr_meulage_bavure_182 := [[58.59753515625,201.009453125,23],[0.999962332692879,-0.00308894112002274,0.00810992655596785,0.000143977181842369],[0,0,0,0],[8.999999E+09,8.999999E+09,8.999999E+09,8.999999E+09,8.999999E+09,8.999999E+09]];
    LOCAL CONST Robtarget Tr_meulage_bavure_183 := [[60.100890625,201.62865625,23],[0.999962813781141,-0.00299887719091118,0.00808413854237589,0.000156507268815584],[0,0,0,0],[8.999999E+09,8.999999E+09,8.999999E+09,8.999999E+09,8.999999E+09,8.999999E+09]];
    LOCAL CONST Robtarget Tr_meulage_bavure_184 := [[62.44671484375,202.59871875,23],[0.999963703838614,-0.00278726356940505,0.00804948868631697,0.000167030070809919],[0,0,0,0],[8.999999E+09,8.999999E+09,8.999999E+09,8.999999E+09,8.999999E+09,8.999999E+09]];
    LOCAL CONST Robtarget Tr_meulage_bavure_185 := [[64.86050390625,203.50121875,23],[0.999965148555411,-0.00239793272775408,0.00799505334554296,0.000175257494603603],[0,0,0,0],[8.999999E+09,8.999999E+09,8.999999E+09,8.999999E+09,8.999999E+09,8.999999E+09]];
    LOCAL CONST Robtarget Tr_meulage_bavure_186 := [[68.275875,204.921234375,23],[0.999967165630264,-0.00178555432269475,0.00790232303327491,0.000180963573031834],[0,0,0,0],[8.999999E+09,8.999999E+09,8.999999E+09,8.999999E+09,8.999999E+09,8.999999E+09]];
    LOCAL CONST Robtarget Tr_meulage_bavure_187 := [[71.1980859375,206.141171875,23],[0.99996957967494,-0.000933169269885203,0.0077417754925405,0.00018393493788852],[0,0,0,0],[8.999999E+09,8.999999E+09,8.999999E+09,8.999999E+09,8.999999E+09,8.999999E+09]];
    LOCAL CONST Robtarget Tr_meulage_bavure_188 := [[72.951328125,206.808015625,23],[0.999972046178929,0.000137669188868629,0.00747353770017586,0.000184775983492988],[0,0,0,0],[8.999999E+09,8.999999E+09,8.999999E+09,8.999999E+09,8.999999E+09,8.999999E+09]];
    LOCAL CONST Robtarget Tr_meulage_bavure_189 := [[75.2215,207.202640625,23],[0.999974151654778,0.00136622091067522,0.00705658579146373,0.000184552699674885],[0,0,0,0],[8.999999E+09,8.999999E+09,8.999999E+09,8.999999E+09,8.999999E+09,8.999999E+09]];
    LOCAL CONST Robtarget Tr_meulage_bavure_190 := [[77.3096640625,207.633734375,23],[0.999975537930332,0.00266691285640391,0.00646351659276342,0.000184580644468813],[0,0,0,0],[8.999999E+09,8.999999E+09,8.999999E+09,8.999999E+09,8.999999E+09,8.999999E+09]];
    LOCAL CONST Robtarget Tr_meulage_bavure_191 := [[79.4188203125,206.551265625,23],[0.999975945369485,0.00394867240108501,0.0056992992608443,0.000186162853842838],[0,0,0,0],[8.999999E+09,8.999999E+09,8.999999E+09,8.999999E+09,8.999999E+09,8.999999E+09]];
    LOCAL CONST Robtarget Tr_meulage_bavure_192 := [[80.0400703125,206.331109375,23],[0.999975242384423,0.00513230337113271,0.00481019631196182,0.000189978319869721],[0,0,0,0],[8.999999E+09,8.999999E+09,8.999999E+09,8.999999E+09,8.999999E+09,8.999999E+09]];
    LOCAL CONST Robtarget Tr_meulage_bavure_193 := [[81.567015625,203.339421875,23],[0.999973492926686,0.00615860089618004,0.00387900311596498,0.000195994464381853],[0,0,0,0],[8.999999E+09,8.999999E+09,8.999999E+09,8.999999E+09,8.999999E+09,8.999999E+09]];
    LOCAL CONST Robtarget Tr_meulage_bavure_194 := [[81.8603828125,202.80884375,23],[0.999971020503959,0.00699295702830144,0.00300255664352445,0.00020336635519608],[0,0,0,0],[8.999999E+09,8.999999E+09,8.999999E+09,8.999999E+09,8.999999E+09,8.999999E+09]];
    LOCAL CONST Robtarget Tr_meulage_bavure_195 := [[81.8648359375,202.806765625,23],[0.999968348867756,0.00762512004091595,0.00226150483646666,0.000210720028629107],[0,0,0,0],[8.999999E+09,8.999999E+09,8.999999E+09,8.999999E+09,8.999999E+09,8.999999E+09]];
    LOCAL CONST Robtarget Tr_meulage_bavure_196 := [[81.9259375,202.649359375,23],[0.999965985066273,0.00806828169922843,0.00169835262128056,0.000217115713540633],[0,0,0,0],[8.999999E+09,8.999999E+09,8.999999E+09,8.999999E+09,8.999999E+09,8.999999E+09]];
    LOCAL CONST Robtarget Tr_meulage_bavure_197 := [[81.9753125,202.195125,23],[0.999964230347926,0.0083524341012969,0.00131363968574065,0.000221855897509995],[0,0,0,0],[8.999999E+09,8.999999E+09,8.999999E+09,8.999999E+09,8.999999E+09,8.999999E+09]];
    LOCAL CONST Robtarget Tr_meulage_bavure_198 := [[82.1716953125,200.726875,23],[0.999963120761309,0.00851753651660019,0.00107616290425912,0.000224860835081592],[0,0,0,0],[8.999999E+09,8.999999E+09,8.999999E+09,8.999999E+09,8.999999E+09,8.999999E+09]];
    LOCAL CONST Robtarget Tr_meulage_bavure_199 := [[82.2009609375,200.3215,23],[0.999962513447803,0.00860410025160748,0.000943381122162763,0.000226252229704601],[0,0,0,0],[8.999999E+09,8.999999E+09,8.999999E+09,8.999999E+09,8.999999E+09,8.999999E+09]];
    LOCAL CONST Robtarget Tr_meulage_bavure_200 := [[82.60821875,195.031796875,23],[0.9999622348982,0.00864347675901973,0.000876315018137209,0.000226183336947231],[0,0,0,0],[8.999999E+09,8.999999E+09,8.999999E+09,8.999999E+09,8.999999E+09,8.999999E+09]];
    LOCAL CONST Robtarget Tr_meulage_bavure_201 := [[83.064609375,189.71584375,23],[0.999962148249332,0.00865640029441431,0.000847470181426941,0.00022493736051429],[0,0,0,0],[8.999999E+09,8.999999E+09,8.999999E+09,8.999999E+09,8.999999E+09,8.999999E+09]];
    LOCAL CONST Robtarget Tr_meulage_bavure_202 := [[83.291078125,186.89309375,23],[0.999962196845362,0.00865110443795112,0.000844844055414829,0.000222510051651043],[0,0,0,0],[8.999999E+09,8.999999E+09,8.999999E+09,8.999999E+09,8.999999E+09,8.999999E+09]];
    LOCAL CONST Robtarget Tr_meulage_bavure_203 := [[83.4083828125,185.326875,23],[0.999962391611422,0.00862635532431872,0.000868043433365498,0.000218762840801778],[0,0,0,0],[8.999999E+09,8.999999E+09,8.999999E+09,8.999999E+09,8.999999E+09,8.999999E+09]];
    LOCAL CONST Robtarget Tr_meulage_bavure_204 := [[83.80996875,181.384953125,23],[0.999962796601448,0.00857300551600752,0.000929153400501553,0.000213689942893135],[0,0,0,0],[8.999999E+09,8.999999E+09,8.999999E+09,8.999999E+09,8.999999E+09,8.999999E+09]];
    LOCAL CONST Robtarget Tr_meulage_bavure_205 := [[84.4078046875,176.141171875,23],[0.999963491979799,0.00847764355901494,0.00104947570051725,0.000207045905800528],[0,0,0,0],[8.999999E+09,8.999999E+09,8.999999E+09,8.999999E+09,8.999999E+09,8.999999E+09]];
    LOCAL CONST Robtarget Tr_meulage_bavure_206 := [[84.74215625,173.671625,23],[0.99996449604871,0.00833153545288826,0.00124605893413982,0.000198736457666264],[0,0,0,0],[8.999999E+09,8.999999E+09,8.999999E+09,8.999999E+09,8.999999E+09,8.999999E+09]];
    LOCAL CONST Robtarget Tr_meulage_bavure_207 := [[84.9359453125,171.51334375,23],[0.999965702417182,0.00814007591683182,0.00151575633398987,0.000188775303899037],[0,0,0,0],[8.999999E+09,8.999999E+09,8.999999E+09,8.999999E+09,8.999999E+09,8.999999E+09]];
    LOCAL CONST Robtarget Tr_meulage_bavure_208 := [[84.9572109375,170.9715,23],[0.999966881463469,0.00793015602405723,0.00182127833483972,0.000177614428669666],[0,0,0,0],[8.999999E+09,8.999999E+09,8.999999E+09,8.999999E+09,8.999999E+09,8.999999E+09]];
    LOCAL CONST Robtarget Tr_meulage_bavure_209 := [[85.00009375,170.01140625,23],[0.999967785675096,0.00774701605462761,0.00209377184874417,0.000165752045643028],[0,0,0,0],[8.999999E+09,8.999999E+09,8.999999E+09,8.999999E+09,8.999999E+09,8.999999E+09]];
    LOCAL CONST Robtarget Tr_meulage_bavure_210 := [[85.3654140625,161.88396875,23],[0.99996826315128,0.00763944214256083,0.00225566690536902,0.000153560329989759],[0,0,0,0],[8.999999E+09,8.999999E+09,8.999999E+09,8.999999E+09,8.999999E+09,8.999999E+09]];
    LOCAL CONST Robtarget Tr_meulage_bavure_211 := [[85.462375,161.8231875,23],[0.999968266135104,0.00763993863137262,0.00225344236050954,0.000141626235167489],[0,0,0,0],[8.999999E+09,8.999999E+09,8.999999E+09,8.999999E+09,8.999999E+09,8.999999E+09]];
    LOCAL CONST Robtarget Tr_meulage_bavure_212 := [[85.6098359375,158.448890625,23],[0.999967797177128,0.00774870936939717,0.00208451038764056,0.000130108699908082],[0,0,0,0],[8.999999E+09,8.999999E+09,8.999999E+09,8.999999E+09,8.999999E+09,8.999999E+09]];
    LOCAL CONST Robtarget Tr_meulage_bavure_213 := [[85.780546875,155.384640625,23],[0.999966904418536,0.00793358554868372,0.00179837513342972,0.00011888999647273],[0,0,0,0],[8.999999E+09,8.999999E+09,8.999999E+09,8.999999E+09,8.999999E+09,8.999999E+09]];
    LOCAL CONST Robtarget Tr_meulage_bavure_214 := [[86.0823984375,149.711453125,23],[0.999965733804557,0.00814598572099555,0.00147054537782019,0.000107840807312128],[0,0,0,0],[8.999999E+09,8.999999E+09,8.999999E+09,8.999999E+09,8.999999E+09,8.999999E+09]];
    LOCAL CONST Robtarget Tr_meulage_bavure_215 := [[86.138578125,148.8935,23],[0.999964526562773,0.0083407192842188,0.0011699032833266,9.66654976046569E-05],[0,0,0,0],[8.999999E+09,8.999999E+09,8.999999E+09,8.999999E+09,8.999999E+09,8.999999E+09]];
    LOCAL CONST Robtarget Tr_meulage_bavure_216 := [[86.470546875,142.730015625,23],[0.999963511709568,0.00849079893068827,0.000935037351269643,8.53706031057797E-05],[0,0,0,0],[8.999999E+09,8.999999E+09,8.999999E+09,8.999999E+09,8.999999E+09,8.999999E+09]];
    LOCAL CONST Robtarget Tr_meulage_bavure_217 := [[86.5939921875,140.929625,23],[0.999962800243306,0.00859061048812701,0.000770753786567553,7.40243730085405E-05],[0,0,0,0],[8.999999E+09,8.999999E+09,8.999999E+09,8.999999E+09,8.999999E+09,8.999999E+09]];
    LOCAL CONST Robtarget Tr_meulage_bavure_218 := [[86.7443515625,139.27765625,23],[0.999962374847901,0.00864912221460549,0.000661533510417842,6.28241750424876E-05],[0,0,0,0],[8.999999E+09,8.999999E+09,8.999999E+09,8.999999E+09,8.999999E+09,8.999999E+09]];
    LOCAL CONST Robtarget Tr_meulage_bavure_219 := [[86.8099375,137.8385,23],[0.999962149960207,0.00868046739435036,0.000587718237090061,5.21540920561728E-05],[0,0,0,0],[8.999999E+09,8.999999E+09,8.999999E+09,8.999999E+09,8.999999E+09,8.999999E+09]];
    LOCAL CONST Robtarget Tr_meulage_bavure_220 := [[86.8993203125,135.272765625,23],[0.99996204568879,0.00869575389268065,0.000537844830675382,4.20602721612032E-05],[0,0,0,0],[8.999999E+09,8.999999E+09,8.999999E+09,8.999999E+09,8.999999E+09,8.999999E+09]];
    LOCAL CONST Robtarget Tr_meulage_bavure_221 := [[86.9025859375,134.49471875,23],[0.999962001896856,0.00870273112696114,0.00050612258452435,3.27611615386615E-05],[0,0,0,0],[8.999999E+09,8.999999E+09,8.999999E+09,8.999999E+09,8.999999E+09,8.999999E+09]];
    LOCAL CONST Robtarget Tr_meulage_bavure_222 := [[86.9266953125,132.059484375,23],[0.999961982050637,0.00870603839535817,0.000488633038918964,2.42192905273249E-05],[0,0,0,0],[8.999999E+09,8.999999E+09,8.999999E+09,8.999999E+09,8.999999E+09,8.999999E+09]];
    LOCAL CONST Robtarget Tr_meulage_bavure_223 := [[86.9136328125,130.817109375,23],[0.999961974338028,0.00870732821524004,0.000481712802728698,1.63132125731158E-05],[0,0,0,0],[8.999999E+09,8.999999E+09,8.999999E+09,8.999999E+09,8.999999E+09,8.999999E+09]];
    LOCAL CONST Robtarget Tr_meulage_bavure_224 := [[86.975953125,129.6813359375,23],[0.999961970448947,0.00870795017706445,0.000478723733578853,9.11920637298542E-06],[0,0,0,0],[8.999999E+09,8.999999E+09,8.999999E+09,8.999999E+09,8.999999E+09,8.999999E+09]];
    LOCAL CONST Robtarget Tr_meulage_bavure_225 := [[87.2295859375,125.4028046875,23],[0.999961966098141,0.00870875759248517,0.000473172864454783,2.40351190441421E-06],[0,0,0,0],[8.999999E+09,8.999999E+09,8.999999E+09,8.999999E+09,8.999999E+09,8.999999E+09]];
    LOCAL CONST Robtarget Tr_meulage_bavure_226 := [[87.3719140625,122.88946875,23],[0.999961961349824,0.00870990810187198,0.000461885873383911,-3.96360151290942E-06],[0,0,0,0],[8.999999E+09,8.999999E+09,8.999999E+09,8.999999E+09,8.999999E+09,8.999999E+09]];
    LOCAL CONST Robtarget Tr_meulage_bavure_227 := [[87.5888671875,120.5894453125,23],[0.999961956427166,0.00871131689719273,0.000445593028892499,-1.01549592746791E-05],[0,0,0,0],[8.999999E+09,8.999999E+09,8.999999E+09,8.999999E+09,8.999999E+09,8.999999E+09]];
    LOCAL CONST Robtarget Tr_meulage_bavure_228 := [[87.7881484375,117.7775859375,23],[0.999961951954065,0.0087126839607579,0.000428378550029935,-1.65599957897006E-05],[0,0,0,0],[8.999999E+09,8.999999E+09,8.999999E+09,8.999999E+09,8.999999E+09,8.999999E+09]];
    LOCAL CONST Robtarget Tr_meulage_bavure_229 := [[88.0114140625,112.2958359375,23],[0.999961948941226,0.00871363125256458,0.000415639822159104,-2.33151823581659E-05],[0,0,0,0],[8.999999E+09,8.999999E+09,8.999999E+09,8.999999E+09,8.999999E+09,8.999999E+09]];
    LOCAL CONST Robtarget Tr_meulage_bavure_230 := [[88.210234375,107.0625,23],[0.999961948356287,0.00871385684889625,0.000411822572903652,-3.06672899654357E-05],[0,0,0,0],[8.999999E+09,8.999999E+09,8.999999E+09,8.999999E+09,8.999999E+09,8.999999E+09]];
    LOCAL CONST Robtarget Tr_meulage_bavure_231 := [[88.36725,103.8018515625,23],[0.999961950560472,0.00871321597682122,0.000419275171645036,-3.88196784471151E-05],[0,0,0,0],[8.999999E+09,8.999999E+09,8.999999E+09,8.999999E+09,8.999999E+09,8.999999E+09]];
    LOCAL CONST Robtarget Tr_meulage_bavure_232 := [[88.4679296875,101.3322734375,23],[0.999961954887377,0.00871177656706648,0.000437532971550119,-4.78723276706944E-05],[0,0,0,0],[8.999999E+09,8.999999E+09,8.999999E+09,8.999999E+09,8.999999E+09,8.999999E+09]];
    LOCAL CONST Robtarget Tr_meulage_bavure_233 := [[88.4963046875,99.366546875,23],[0.999961959881839,0.00870979527769241,0.00046357360963568,-5.79223635319835E-05],[0,0,0,0],[8.999999E+09,8.999999E+09,8.999999E+09,8.999999E+09,8.999999E+09,8.999999E+09]];
    LOCAL CONST Robtarget Tr_meulage_bavure_234 := [[88.8017890625,96.0728125,23],[0.999961963929494,0.00870765641443032,0.000492630648860709,-6.87683169445721E-05],[0,0,0,0],[8.999999E+09,8.999999E+09,8.999999E+09,8.999999E+09,8.999999E+09,8.999999E+09]];
    LOCAL CONST Robtarget Tr_meulage_bavure_235 := [[88.92840625,93.9544375,23],[0.999961965899355,0.0087057811337698,0.000519275568681911,-8.05135532927361E-05],[0,0,0,0],[8.999999E+09,8.999999E+09,8.999999E+09,8.999999E+09,8.999999E+09,8.999999E+09]];
    LOCAL CONST Robtarget Tr_meulage_bavure_236 := [[89.0796484375,92.279390625,23],[0.999961965371174,0.00870453830115365,0.000538662916731642,-9.30926692764098E-05],[0,0,0,0],[8.999999E+09,8.999999E+09,8.999999E+09,8.999999E+09,8.999999E+09,8.999999E+09]];
    LOCAL CONST Robtarget Tr_meulage_bavure_237 := [[89.1046171875,91.3662734375,23],[0.999961962472182,0.00870415091639765,0.000547801452269028,-0.000106203468209855],[0,0,0,0],[8.999999E+09,8.999999E+09,8.999999E+09,8.999999E+09,8.999999E+09,8.999999E+09]];
    LOCAL CONST Robtarget Tr_meulage_bavure_238 := [[89.1337578125,90.875515625,23],[0.999961957453897,0.00870462951427438,0.000546537153629104,-0.000119862963017372],[0,0,0,0],[8.999999E+09,8.999999E+09,8.999999E+09,8.999999E+09,8.999999E+09,8.999999E+09]];
    LOCAL CONST Robtarget Tr_meulage_bavure_239 := [[89.16028125,89.797359375,23],[0.999961950670275,0.00870578092470559,0.000537256792385921,-0.000133960176885578],[0,0,0,0],[8.999999E+09,8.999999E+09,8.999999E+09,8.999999E+09,8.999999E+09,8.999999E+09]];
    LOCAL CONST Robtarget Tr_meulage_bavure_240 := [[89.189546875,88.7360546875,23],[0.999961942713709,0.00870726299156617,0.000524128348852551,-0.000148273044481476],[0,0,0,0],[8.999999E+09,8.999999E+09,8.999999E+09,8.999999E+09,8.999999E+09,8.999999E+09]];
    LOCAL CONST Robtarget Tr_meulage_bavure_241 := [[89.5481875,80.2841171875,23],[0.99996193465141,0.00870869329025639,0.000511311401804819,-0.000162696145656232],[0,0,0,0],[8.999999E+09,8.999999E+09,8.999999E+09,8.999999E+09,8.999999E+09,8.999999E+09]];
    LOCAL CONST Robtarget Tr_meulage_bavure_242 := [[89.623140625,79.6325390625,23],[0.999961928057909,0.00870972891220971,0.000501722484395105,-0.000177007155121191],[0,0,0,0],[8.999999E+09,8.999999E+09,8.999999E+09,8.999999E+09,8.999999E+09,8.999999E+09]];
    LOCAL CONST Robtarget Tr_meulage_bavure_243 := [[89.6957421875,78.3010859375,23],[0.999961924681602,0.00871014381590187,0.000496046061761808,-0.000191102269185484],[0,0,0,0],[8.999999E+09,8.999999E+09,8.999999E+09,8.999999E+09,8.999999E+09,8.999999E+09]];
    LOCAL CONST Robtarget Tr_meulage_bavure_244 := [[89.6254609375,77.276578125,23],[0.999961926524518,0.00870981854452266,0.000492662549210655,-0.000204562727657816],[0,0,0,0],[8.999999E+09,8.999999E+09,8.999999E+09,8.999999E+09,8.999999E+09,8.999999E+09]];
    LOCAL CONST Robtarget Tr_meulage_bavure_245 := [[89.64715625,76.986359375,23],[0.999961935663691,0.0087086750313148,0.000488935868943349,-0.00021712816461049],[0,0,0,0],[8.999999E+09,8.999999E+09,8.999999E+09,8.999999E+09,8.999999E+09,8.999999E+09]];
    LOCAL CONST Robtarget Tr_meulage_bavure_246 := [[89.7738671875,75.3290703125,23],[0.999961953987859,0.00870666475913039,0.000481911730109789,-0.000228750168392484],[0,0,0,0],[8.999999E+09,8.999999E+09,8.999999E+09,8.999999E+09,8.999999E+09,8.999999E+09]];
    LOCAL CONST Robtarget Tr_meulage_bavure_247 := [[90.246125,69.478640625,23],[0.999961982699416,0.00870378740656149,0.000469158243504417,-0.000239021287849803],[0,0,0,0],[8.999999E+09,8.999999E+09,8.999999E+09,8.999999E+09,8.999999E+09,8.999999E+09]];
    LOCAL CONST Robtarget Tr_meulage_bavure_248 := [[90.38025,67.148953125,23],[0.999962021135001,0.00870014968135541,0.000449798185040133,-0.000247719029854836],[0,0,0,0],[8.999999E+09,8.999999E+09,8.999999E+09,8.999999E+09,8.999999E+09,8.999999E+09]];
    LOCAL CONST Robtarget Tr_meulage_bavure_249 := [[90.570921875,58.42654296875,23],[0.999962066277403,0.00869600918925303,0.000424859399085087,-0.000254803646331772],[0,0,0,0],[8.999999E+09,8.999999E+09,8.999999E+09,8.999999E+09,8.999999E+09,8.999999E+09]];
    LOCAL CONST Robtarget Tr_meulage_bavure_250 := [[90.6774609375,54.2451171875,23],[0.999962112802246,0.00869176989311296,0.000398007636375098,-0.000260165552805419],[0,0,0,0],[8.999999E+09,8.999999E+09,8.999999E+09,8.999999E+09,8.999999E+09,8.999999E+09]];
    LOCAL CONST Robtarget Tr_meulage_bavure_251 := [[90.73190625,52.53121875,23],[0.999962154449225,0.0086878409134516,0.000376165394959878,-0.00026379750219836],[0,0,0,0],[8.999999E+09,8.999999E+09,8.999999E+09,8.999999E+09,8.999999E+09,8.999999E+09]];
    LOCAL CONST Robtarget Tr_meulage_bavure_252 := [[91.2394375,46.3190625,23],[0.999962185784896,0.00868451235850285,0.000368298759695558,-0.000265709260958138],[0,0,0,0],[8.999999E+09,8.999999E+09,8.999999E+09,8.999999E+09,8.999999E+09,8.999999E+09]];
    LOCAL CONST Robtarget Tr_meulage_bavure_253 := [[91.37384375,44.75738671875,23],[0.999962203038616,0.0086819045323968,0.000382430890160427,-0.000266034699544847],[0,0,0,0],[8.999999E+09,8.999999E+09,8.999999E+09,8.999999E+09,8.999999E+09,8.999999E+09]];
    LOCAL CONST Robtarget Tr_meulage_bavure_254 := [[91.413515625,44.36984375,23],[0.99996220403107,0.00867998554383968,0.000422148994740198,-0.000264859417002956],[0,0,0,0],[8.999999E+09,8.999999E+09,8.999999E+09,8.999999E+09,8.999999E+09,8.999999E+09]];
    LOCAL CONST Robtarget Tr_meulage_bavure_255 := [[91.416046875,44.01062109375,23],[0.999962188262155,0.00867861034368897,0.000484739830256208,-0.000262289461304777],[0,0,0,0],[8.999999E+09,8.999999E+09,8.999999E+09,8.999999E+09,8.999999E+09,8.999999E+09]];
    LOCAL CONST Robtarget Tr_meulage_bavure_256 := [[92.0011015625,39.38336328125,23],[0.999962158118112,0.0086775936395806,0.000561210084705216,-0.000258347897461707],[0,0,0,0],[8.999999E+09,8.999999E+09,8.999999E+09,8.999999E+09,8.999999E+09,8.999999E+09]];
    LOCAL CONST Robtarget Tr_meulage_bavure_257 := [[92.1544765625,37.63262890625,23],[0.999962119694029,0.00867673604529358,0.000639823354867034,-0.000253090298893801],[0,0,0,0],[8.999999E+09,8.999999E+09,8.999999E+09,8.999999E+09,8.999999E+09,8.999999E+09]];
    LOCAL CONST Robtarget Tr_meulage_bavure_258 := [[92.331265625,33.3674609375,23],[0.999962081756606,0.00867590204294796,0.000709194072541833,-0.000246610024303043],[0,0,0,0],[8.999999E+09,8.999999E+09,8.999999E+09,8.999999E+09,8.999999E+09,8.999999E+09]];
